(* PLC project fablewhole, LeadShine company LeadSys Studio V3.1.0.0 LeadSysStudio V3.5 SP15 Patch 4 *)
(* stored: creationDateTime 2026-07-10T18:08:29.5976327, modificationDateTime 2026-07-10T18:07:30.2023087 *)

{attribute 'qualified_only'}
{attribute 'strict'}
TYPE E_MachMode : (BOOT := 0, HOMING := 1, READY := 2, RUN := 3, CLEAN := 4, FAULT := 5, ESTOP := 6);
END_TYPE

{attribute 'qualified_only'}
{attribute 'strict'}
TYPE E_Item : (NONE := 0, BEEF := 1, CHICKEN := 2, BACON := 3, PINEAPPLE := 4);
END_TYPE

{attribute 'qualified_only'}
{attribute 'strict'}
TYPE E_GriddleState : (EMPTY := 0, LOADING := 1, COOKING := 2, READY_TO_SCRAPE := 3, SCRAPING := 4, FAULTED := 5);
END_TYPE

{attribute 'qualified_only'}
{attribute 'strict'}
TYPE E_FaultClass : (INFO := 0, QUARANTINE := 1, ZONE_STOP := 2, MACHINE_STOP := 3);
END_TYPE

TYPE ST_Recipe : STRUCT
  item : UINT;  (* E_Item value *)
  cookTimeS : LREAL := 90.0;
  smashDurS : LREAL := 8.0;
  smashPosMm : LREAL := 4.0;  (* platen gap at smash *)
  holdPosMm : LREAL := 6.0;  (* light-contact gap for remainder of cook *)
  platenSetC : LREAL := 200.0;
END_STRUCT;
END_TYPE

TYPE ST_PattyJob : STRUCT
  jobId : UDINT;
  orderId : UDINT;
  item : UINT;
  trayId : UINT;
  griddleId : INT;
  slot : INT;
END_STRUCT;
END_TYPE

TYPE ST_GriddleSts : STRUCT
  state : UINT;  (* E_GriddleState value *)
  item : UINT;
  count : INT;
  cookElapsedS : LREAL;
  batchId : UDINT;
END_STRUCT;
END_TYPE

TYPE ST_TrayInfo : STRUCT
  trayId : UINT;
  item : UINT;
  remaining : INT;
  level : INT;  (* 0..19 *)
  face : INT;  (* 0..1 *)
  inChamber : BOOL;
END_STRUCT;
END_TYPE

TYPE ST_GwCmd : STRUCT
  seq : UINT;
  code : UINT;  (* see GVL_Cfg CMD_* constants *)
  p1 : DINT;
  p2 : DINT;
  p3 : DINT;
  p4 : DINT;
END_STRUCT;
END_TYPE

TYPE ST_GwAck : STRUCT
  seqEcho : UINT;
  busy : BOOL;
  done : BOOL;
  error : BOOL;
  errorId : UDINT;
END_STRUCT;
END_TYPE

TYPE ST_AxisSts : STRUCT
  powered : BOOL;
  homed : BOOL;
  inPos : BOOL;
  actPos : LREAL;
  errorId : UDINT;
END_STRUCT;
END_TYPE

TYPE ST_HeatZone : STRUCT
  setC : LREAL;
  actC : LREAL;
  outPct : LREAL;
  tcOk : BOOL;
  atSet : BOOL;
  enabled : BOOL;
END_STRUCT;
END_TYPE

TYPE ST_Alarm : STRUCT
  id : UDINT;  (* (subsystem<<16) OR code *)
  class : UINT;  (* E_FaultClass value *)
  tsS : UDINT;  (* uptime seconds at raise *)
  active : BOOL;
  acked : BOOL;
END_STRUCT;
END_TYPE

TYPE ST_HaccpRec : STRUCT
  batchId : UDINT;
  item : UINT;
  griddleId : INT;
  platenTopC : LREAL;
  platenBotC : LREAL;
  cookS : LREAL;
  tStartS : UDINT;
  tEndS : UDINT;
  result : UINT;  (* 0=OK 1=QUARANTINE *)
END_STRUCT;
END_TYPE

TYPE ST_MechCmd : STRUCT
  code : UINT;  (* mechanism-local, see GVL_Cfg MCMD_* constants *)
  p1 : LREAL;
  p2 : LREAL;
  p3 : LREAL;
END_STRUCT;
END_TYPE

(* ===== FUNCTION F_Err : UDINT ===== ErrorID encoding: (subsystem << 16) OR code *)
FUNCTION F_Err : UDINT
  VAR_INPUT
    ss : UINT;
    code : UINT;
  END_VAR

                    F_Err := SHL(TO_UDINT(ss), 16) OR TO_UDINT(code);

                  
END_FUNCTION

(* ===== FUNCTION F_RaiseAlarm : BOOL ===== Latch an alarm into GVL_Alm (dedup by id). Returns TRUE if new. *)
FUNCTION F_RaiseAlarm : BOOL
  VAR_INPUT
    id : UDINT;
    class : UINT;  (* E_FaultClass value *)
  END_VAR
  VAR
    i : INT;
  END_VAR

                    F_RaiseAlarm := FALSE;
IF id = 0 THEN RETURN; END_IF
FOR i := 0 TO 63 DO
    IF GVL_Alm.aActive[i].active AND (GVL_Alm.aActive[i].id = id) THEN
        RETURN;                      // already active
    END_IF
END_FOR
FOR i := 0 TO 63 DO
    IF NOT GVL_Alm.aActive[i].active THEN
        GVL_Alm.aActive[i].id     := id;
        GVL_Alm.aActive[i].class  := class;
        GVL_Alm.aActive[i].tsS    := GVL_Sts.uptimeS;
        GVL_Alm.aActive[i].active := TRUE;
        GVL_Alm.aActive[i].acked  := FALSE;
        // history ring
        GVL_Alm.aHistory[GVL_Alm.histHead] := GVL_Alm.aActive[i];
        GVL_Alm.histHead := (GVL_Alm.histHead + 1) MOD 200;
        F_RaiseAlarm := TRUE;
        RETURN;
    END_IF
END_FOR


                  
END_FUNCTION

(* ============================================================ FB_AxisCtrl — single-axis wrapper. The ONLY POU calling MC_*. Runs in T_Motion. One instance per axis, body called EVERY cycle. SIM: internal kinematic model (trapezoid-less: const-vel ramp). REAL: SoftMotion CiA-402 via SM3_Basic. ============================================================ *)
FUNCTION_BLOCK FB_AxisCtrl
  VAR_INPUT
    Sim : BOOL;
    SubsysId : UINT;
    Enable : BOOL;
    HomeExec : BOOL;  (* level; internally edge-latched *)
    MoveExec : BOOL;
    TargetPos : LREAL;
    Vel : LREAL := 100.0;
    Acc : LREAL := 500.0;
    StopExec : BOOL;
    ResetExec : BOOL;
    Abort : BOOL;
    CycleMs : LREAL := 4.0;
    SimHomeS : LREAL := 1.0;  (* sim homing duration *)
  END_VAR
  VAR_IN_OUT
    Axis : AXIS_REF_SM3;
  END_VAR
  VAR_OUTPUT
    Sts : ST_AxisSts;
    Busy : BOOL;
    Done : BOOL;  (* latched until next exec *)
    Error : BOOL;
    ErrorID : UDINT;
  END_VAR
  VAR
    state : INT;  (* 0 idle 1 homing 2 moving 3 stopping *)
    rtHome : R_TRIG;
    rtMove : R_TRIG;
    rtReset : R_TRIG;
    tonTO : TON;
    simPos : LREAL;  (* sim model *)
    simTgt : LREAL;
    simHomeT : LREAL;
    mcPower : MC_Power;  (* real motion FBs *)
    mcHome : MC_Home;
    mcMove : MC_MoveAbsolute;
    mcStop : MC_Stop;
    mcReset : MC_Reset;
    dtS : LREAL;
    stepMax : LREAL;
  END_VAR

                    
dtS := CycleMs / 1000.0;
rtHome(CLK := HomeExec);
rtMove(CLK := MoveExec);
rtReset(CLK := ResetExec);

IF Abort THEN
    state := 0; Busy := FALSE;
    tonTO(IN := FALSE);
END_IF

IF rtReset.Q THEN
    Error := FALSE; ErrorID := 0;
END_IF

IF Sim THEN
    // ---------------- SIMULATION MODEL ----------------
    Sts.powered := Enable;
    CASE state OF
        0: // idle
            IF Enable AND rtHome.Q THEN
                state := 1; simHomeT := 0.0; Busy := TRUE; Done := FALSE;
            ELSIF Enable AND Sts.homed AND rtMove.Q THEN
                simTgt := TargetPos; state := 2; Busy := TRUE; Done := FALSE;
                tonTO(IN := FALSE);
            ELSIF Enable AND (NOT Sts.homed) AND rtMove.Q THEN
                Error := TRUE; ErrorID := F_Err(SubsysId, GVL_Cfg.ERR_NOT_HOMED);
            END_IF
        1: // homing
            simHomeT := simHomeT + dtS;
            IF simHomeT >= SimHomeS THEN
                simPos := 0.0; Sts.homed := TRUE;
                state := 0; Busy := FALSE; Done := TRUE;
            END_IF
        2: // moving: constant-velocity approach
            stepMax := Vel * dtS;
            IF ABS(simTgt - simPos) <= stepMax THEN
                simPos := simTgt;
                state := 0; Busy := FALSE; Done := TRUE;
            ELSIF simTgt > simPos THEN
                simPos := simPos + stepMax;
            ELSE
                simPos := simPos - stepMax;
            END_IF
            tonTO(IN := TRUE, PT := GVL_Cfg.TO_AXIS_MOVE);
            IF tonTO.Q THEN
                state := 0; Busy := FALSE; Error := TRUE;
                ErrorID := F_Err(SubsysId, GVL_Cfg.ERR_TIMEOUT);
            END_IF
    END_CASE
    IF StopExec THEN state := 0; Busy := FALSE; END_IF
    Sts.actPos := simPos;
    Sts.inPos  := (state = 0);
ELSE
    // ---------------- REAL HARDWARE (SoftMotion) ----------------
    mcPower(Axis := Axis, Enable := Enable, bRegulatorOn := Enable, bDriveStart := Enable);
    Sts.powered := mcPower.Status;

    mcHome(Axis := Axis, Execute := (rtHome.Q OR mcHome.Busy) AND NOT Abort, Position := 0.0);
    IF mcHome.Done THEN Sts.homed := TRUE; END_IF

    mcMove(Axis := Axis,
           Execute      := (rtMove.Q OR mcMove.Busy) AND NOT Abort AND NOT StopExec,
           Position     := TargetPos,
           Velocity     := Vel,
           Acceleration := Acc,
           Deceleration := Acc);

    mcStop(Axis := Axis, Execute := StopExec OR Abort, Deceleration := Acc * 2.0);
    mcReset(Axis := Axis, Execute := rtReset.Q);

    Busy := mcHome.Busy OR mcMove.Busy;
    IF mcHome.Done OR mcMove.Done THEN Done := TRUE; END_IF
    IF rtHome.Q OR rtMove.Q THEN Done := FALSE; END_IF

    IF mcMove.Error OR mcHome.Error OR mcPower.Error THEN
        Error := TRUE;
        ErrorID := F_Err(SubsysId, GVL_Cfg.ERR_DRIVE);
        Sts.homed := FALSE;              // demand re-home after drive fault
    END_IF
    Sts.actPos := Axis.fSetPosition;     // TODO: use MC_ReadActualPosition if preferred
    Sts.inPos  := NOT Busy;
END_IF

IF NOT Sts.powered THEN Sts.homed := FALSE; END_IF   // power loss clears homed
Sts.errorId := ErrorID;


                  
END_FUNCTION_BLOCK

(* ============================================================ FB_PidHeater — PI + time-proportioned SSR + TC plausibility. Call every T_App cycle; internal divider executes PI at 100 ms. SIM: first-order plant dT = (gain*out - (T-Tamb)/tau) * dt Independent hardwired thermostat is the REAL protection; the over-temp check here is early warning (INFO/ZONE only). ============================================================ *)
FUNCTION_BLOCK FB_PidHeater
  VAR_INPUT
    Sim : BOOL;
    ZoneId : INT;  (* 0..7 *)
    Enable : BOOL;
    SetC : LREAL := 200.0;
    iTempRaw : INT;  (* 0.1 degC from TC module *)
    StaggerToken : BOOL;  (* may ramp (from FB_HeatBank) *)
    CycleMs : LREAL := 20.0;
  END_VAR
  VAR_OUTPUT
    qSsr : BOOL;
    Zone : ST_HeatZone;
    Error : BOOL;
    ErrorID : UDINT;
  END_VAR
  VAR
    divCnt : INT;
    actC : LREAL;
    lastC : LREAL;
    err : LREAL;
    integ : LREAL;
    outPct : LREAL;
    pwmT : LREAL;
    simC : LREAL := 25.0;
    dtPi : LREAL := 0.1;
    tcFaultCnt : INT;
    SIM_GAIN : LREAL := 3.5;  (* degC/s at 100 % *)
    SIM_TAU : LREAL := 60.0;
    ramping : BOOL;
  END_VAR

                    // ---- acquire temperature ----
IF Sim THEN
    simC := simC + (SIM_GAIN * outPct / 100.0 - (simC - 25.0) / SIM_TAU)
                 * (CycleMs / 1000.0) * GVL_Cfg.SIM_TIME_SCALE;
    actC := simC;
ELSE
    actC := TO_LREAL(iTempRaw) / 10.0;
END_IF

// ---- TC plausibility (real only) ----
IF NOT Sim THEN
    IF (actC < -20.0) OR (actC > 400.0) THEN tcFaultCnt := tcFaultCnt + 1; ELSE tcFaultCnt := 0; END_IF
    IF ABS(actC - lastC) > GVL_Cfg.TC_RATE_MAX * (CycleMs / 1000.0) * 10.0 THEN
        tcFaultCnt := tcFaultCnt + 1;
    END_IF
    IF tcFaultCnt > 25 THEN
        Error := TRUE;
        ErrorID := F_Err(GVL_Cfg.SS_HEAT_0 + TO_UINT(ZoneId), GVL_Cfg.ERR_TC);
    END_IF
END_IF
lastC := actC;

// ---- PI @100 ms ----
divCnt := divCnt + 1;
IF divCnt >= 5 THEN
    divCnt := 0;
    ramping := (SetC - actC) > 20.0;
    IF Enable AND NOT Error AND (StaggerToken OR NOT ramping) THEN
        err := SetC - actC;
        integ := LIMIT(0.0, integ + err * GVL_Cfg.HEAT_KI * dtPi * 100.0, 100.0);
        outPct := LIMIT(0.0, GVL_Cfg.HEAT_KP * err + integ, 100.0);
    ELSE
        outPct := 0.0; integ := 0.0;
    END_IF
END_IF

// ---- time-proportioned SSR ----
pwmT := pwmT + CycleMs;
IF pwmT >= GVL_Cfg.PWM_WINDOW_MS THEN pwmT := 0.0; END_IF
qSsr := Enable AND NOT Error AND (pwmT < outPct / 100.0 * GVL_Cfg.PWM_WINDOW_MS);

Zone.setC := SetC;   Zone.actC := actC;   Zone.outPct := outPct;
Zone.tcOk := NOT Error;
Zone.atSet := ABS(SetC - actC) <= GVL_Cfg.HEAT_AT_BAND;
Zone.enabled := Enable;


                  
END_FUNCTION_BLOCK

(* ============================================================ FB_PneuActuator — valve + 2 reed/prox sensors + timeout. Cmd TRUE = extend/open, FALSE = retract/close. Runs in T_App. SIM: sensors flip after SIM_TRAVEL_S. ============================================================ *)
FUNCTION_BLOCK FB_PneuActuator
  VAR_INPUT
    Sim : BOOL;
    SubsysId : UINT;
    Cmd : BOOL;
    iExtended : BOOL;
    iRetracted : BOOL;
    CycleMs : LREAL := 20.0;
  END_VAR
  VAR_OUTPUT
    qValve : BOOL;
    Extended : BOOL;
    Retracted : BOOL;
    Moving : BOOL;
    Error : BOOL;
    ErrorID : UDINT;
  END_VAR
  VAR
    tonTO : TON;
    lastCmd : BOOL;
    simT : LREAL;
    simExt : BOOL;
    SIM_TRAVEL_S : LREAL := 0.3;
    extEff : BOOL;
    retEff : BOOL;
  END_VAR

                    
qValve := Cmd;
IF Cmd <> lastCmd THEN
    simT := 0.0;
    lastCmd := Cmd;
END_IF

IF Sim THEN
    simT := simT + CycleMs / 1000.0;
    IF simT >= SIM_TRAVEL_S THEN simExt := Cmd; END_IF
    extEff := simExt;  retEff := NOT simExt;
ELSE
    extEff := iExtended; retEff := iRetracted;
END_IF

IF extEff AND retEff THEN                 // both sensors -> wiring fault
    Error := TRUE; ErrorID := F_Err(SubsysId, GVL_Cfg.ERR_SENSOR);
END_IF

Extended  := extEff AND NOT retEff;
Retracted := retEff AND NOT extEff;
Moving    := NOT Extended AND NOT Retracted;

tonTO(IN := (Cmd AND NOT Extended) OR (NOT Cmd AND NOT Retracted), PT := GVL_Cfg.TO_PNEU);
IF tonTO.Q THEN
    Error := TRUE; ErrorID := F_Err(SubsysId, GVL_Cfg.ERR_TIMEOUT);
END_IF


                  
END_FUNCTION_BLOCK

(* ============================================================ FB_PressDrive — CS2RS in PR mode, DI-trigger control. Validated pattern from the gantry test project: - set path-select DOs, wait one cycle, raise CTRG and HOLD it until InPos confirms (never a single-scan pulse) - InPos handshake = "saw moving" (InPos drops, then returns) Modbus RTU monitoring (position/alarm) is DIAGNOSTIC ONLY and added at migration (stub hooks below). Runs in T_App (20 ms). PR paths (configure in drive, MIGRATION_GUIDE step 4): path 0 = OPEN position, path 1 = SMASH pos, path 2 = HOLD pos ============================================================ *)
FUNCTION_BLOCK FB_PressDrive
  VAR_INPUT
    Sim : BOOL;
    SubsysId : UINT;
    Enable : BOOL;
    PathExec : BOOL;  (* edge latches PathNo *)
    PathNo : INT;  (* 0..2 *)
    Abort : BOOL;
    iInPos : BOOL;  (* from drive DO (via IoMap) *)
    iAlarm : BOOL;
    CycleMs : LREAL := 20.0;
    OpenPosMm : LREAL := 60.0;  (* path 0 *)
    SmashPosMm : LREAL := 4.0;  (* path 1 *)
    HoldPosMm : LREAL := 6.0;  (* path 2 *)
    WriteParams : BOOL;  (* edge: push the 3 positions to the drive *)
    MbWrDone : BOOL;  (* transport confirms last write *)
    MbWrErr : BOOL;  (* transport reports failure *)
  END_VAR
  VAR_OUTPUT
    qSel0 : BOOL;
    qSel1 : BOOL;
    qCtrg : BOOL;
    qEnable : BOOL;
    Busy : BOOL;
    Done : BOOL;
    Error : BOOL;
    ErrorID : UDINT;
    ActPath : INT := -1;
    ParamsValid : BOOL;  (* drive path table matches last written values *)
    ParamBusy : BOOL;
    ParamErr : BOOL;
    MbPath : INT;  (* which PR path's position is being written (0..2) *)
    MbValH : WORD;  (* position high word *)
    MbValL : WORD;  (* position low word *)
    MbWrExec : BOOL;  (* held TRUE until MbWrDone/MbWrErr *)
  END_VAR
  VAR
    state : INT;
    rtExec : R_TRIG;
    latched : INT;
    sawMoving : BOOL;
    tonTO : TON;
    inPosEff : BOOL;
    simTimer : LREAL;  (* sim *)
    SIM_TRAVEL_S : LREAL := 0.8;
    rtWr : R_TRIG;  (* param write channel *)
    pStep : INT;
    pRetry : INT;
    P_MAX_RETRY : INT := 3;
    shadowOpen : LREAL;  (* last values confirmed in drive *)
    shadowSmash : LREAL;  (* last values confirmed in drive *)
    shadowHold : LREAL;  (* last values confirmed in drive *)
    pInit : BOOL;  (* at least one successful full push done *)
    pIdx : INT;  (* 0..2: one write per PR path (posH+posL together) *)
    pPosMm : LREAL;
    pPulses : DINT;
    tonMb : TON;  (* per-transaction timeout *)
  END_VAR

                    rtExec(CLK := PathExec);
qEnable := Enable;

// effective InPos: sim model or hardware input
IF Sim THEN
    inPosEff := (state <> 3) OR (simTimer >= SIM_TRAVEL_S);
ELSE
    inPosEff := iInPos;
END_IF

IF Abort THEN
    state := 0; Busy := FALSE; qCtrg := FALSE;
    tonTO(IN := FALSE);
END_IF

IF (NOT Sim) AND iAlarm THEN
    Error := TRUE; ErrorID := F_Err(SubsysId, GVL_Cfg.ERR_DRIVE);
    state := 0; Busy := FALSE; qCtrg := FALSE;
    pInit := FALSE;   // drive may have power-cycled: RAM PR table reverts to
                      // EEPROM, so force a full re-push on the next profile
END_IF

CASE state OF
    0: // idle
        qCtrg := FALSE;
        IF Enable AND rtExec.Q AND (PathNo >= 0) AND (PathNo <= 2) THEN
            latched := PathNo;
            qSel0 := (latched MOD 2) = 1;
            qSel1 := ((latched / 2) MOD 2) = 1;
            state := 1; Busy := TRUE; Done := FALSE;
            sawMoving := FALSE; simTimer := 0.0;
            tonTO(IN := FALSE);
        END_IF
    1: // one full cycle DO settle before CTRG (drive DI filter)
        state := 3;
        qCtrg := TRUE;                     // held high for whole move
    3: // executing: wait saw-moving handshake
        simTimer := simTimer + CycleMs / 1000.0;
        IF NOT inPosEff THEN sawMoving := TRUE; END_IF
        tonTO(IN := TRUE, PT := GVL_Cfg.TO_PRESS);
        IF inPosEff AND (sawMoving OR (Sim AND simTimer >= SIM_TRAVEL_S)) THEN
            qCtrg := FALSE; ActPath := latched;
            state := 0; Busy := FALSE; Done := TRUE;
            tonTO(IN := FALSE);
        ELSIF tonTO.Q THEN
            qCtrg := FALSE;
            state := 0; Busy := FALSE; Error := TRUE;
            ErrorID := F_Err(SubsysId, GVL_Cfg.ERR_TIMEOUT);
        END_IF
END_CASE

// ============================================================
// PR path table parameter writer (positions only; motion stays DI).
// SIM: accepted instantly. HARDWARE: closed-loop Modbus RTU write ->
// readback verify -> retry (pattern proven on the old Z-axis rig).
// Only call while press idle; FB_Press guarantees this.
// ============================================================
rtWr(CLK := WriteParams);
IF rtWr.Q AND (pStep = 0) THEN
    ParamsValid := FALSE; ParamErr := FALSE; ParamBusy := TRUE;
    pRetry := 0; pStep := 1;
END_IF

CASE pStep OF
    0: ;
    1: // route: skip if drive already holds these values
        IF pInit AND (OpenPosMm = shadowOpen) AND (SmashPosMm = shadowSmash)
                 AND (HoldPosMm = shadowHold) THEN
            ParamsValid := TRUE; ParamBusy := FALSE; pStep := 0;
        ELSIF Sim THEN
            // simulation: accept instantly
            shadowOpen := OpenPosMm; shadowSmash := SmashPosMm; shadowHold := HoldPosMm;
            pInit := TRUE;
            ParamsValid := TRUE; ParamBusy := FALSE; pStep := 0;
        ELSE
            pIdx := 0; pStep := 2;                        // real Modbus push, path by path
        END_IF
    2: // compose path write pIdx (posH+posL in one write-multiple transaction)
        CASE pIdx OF
            0: pPosMm := OpenPosMm;
            1: pPosMm := SmashPosMm;
            2: pPosMm := HoldPosMm;
        END_CASE
        pPulses := TO_DINT(pPosMm * GVL_Cfg.PRESS_PULSES_PER_MM);
        MbPath := pIdx;
        MbValH := TO_WORD(SHR(TO_DWORD(pPulses), 16) AND 16#FFFF);
        MbValL := TO_WORD(TO_DWORD(pPulses) AND 16#FFFF);
        MbWrExec := TRUE; tonMb(IN := FALSE);
        pStep := 3;
    3: // wait channel ack (glue reflects the NetworkConfig channel done/error)
        tonMb(IN := TRUE, PT := T#1S);
        IF MbWrDone THEN
            MbWrExec := FALSE; tonMb(IN := FALSE); pRetry := 0;
            pIdx := pIdx + 1;
            IF pIdx > 2 THEN
                shadowOpen := OpenPosMm; shadowSmash := SmashPosMm; shadowHold := HoldPosMm;
                pInit := TRUE;
                ParamsValid := TRUE; ParamBusy := FALSE; pStep := 0;
            ELSE
                pStep := 2;                               // next path (fresh trigger edge)
            END_IF
        ELSIF MbWrErr OR tonMb.Q THEN
            MbWrExec := FALSE; tonMb(IN := FALSE);
            pRetry := pRetry + 1;
            IF pRetry > P_MAX_RETRY THEN
                ParamErr := TRUE; ParamBusy := FALSE; pStep := 0;
            ELSE
                pStep := 2;                               // resend same path
            END_IF
        END_IF
END_CASE

// TODO(MIGRATION): background Modbus RTU poll <=2 Hz for ActPosMm +
// AlarmCode; failure raises INFO alarm only, never blocks motion.

                  
END_FUNCTION_BLOCK

(* ============================================================ FB_SensorIn — debounced digital input. SIM: output follows SimValue directly. ============================================================ *)
FUNCTION_BLOCK FB_SensorIn
  VAR_INPUT
    Sim : BOOL;
    SimValue : BOOL;
    iRaw : BOOL;
    DebounceMs : LREAL := 40.0;
    CycleMs : LREAL := 20.0;
  END_VAR
  VAR_OUTPUT
    Q : BOOL;
  END_VAR
  VAR
    acc : LREAL;
    lastRaw : BOOL;
  END_VAR

                    IF Sim THEN
    Q := SimValue;
ELSE
    IF iRaw = lastRaw THEN
        acc := acc + CycleMs;
        IF acc >= DebounceMs THEN Q := iRaw; END_IF
    ELSE
        acc := 0.0;
        lastRaw := iRaw;
    END_IF
END_IF


                  
END_FUNCTION_BLOCK

(* ============================================================ FB_VfdIndex — carousel indexing: VFD run/dir + encoder + pin. Pin actuator is external (FB_PneuActuator); this FB commands it via PinCmd and reads PinExtended/PinRetracted. Sequence: retract pin -> rotate (fast->creep) -> stop in window -> extend pin -> verify pin + encoder plausibility. Runs in T_App. SIM: integrates encoder; home prox modeled. ============================================================ *)
FUNCTION_BLOCK FB_VfdIndex
  VAR_INPUT
    Sim : BOOL;
    SubsysId : UINT;
    Enable : BOOL;
    HomeExec : BOOL;
    GotoExec : BOOL;
    TargetStation : INT;
    Bidirectional : BOOL;
    Abort : BOOL;
    iEnc : DINT;
    iHomeProx : BOOL;
    PinExtended : BOOL;
    PinRetracted : BOOL;
    CycleMs : LREAL := 20.0;
  END_VAR
  VAR_OUTPUT
    qFwd : BOOL;
    qRev : BOOL;
    qSpeed : INT;
    PinCmd : BOOL := TRUE;  (* TRUE = extend (locked at rest) *)
    ActStation : INT := -1;
    Homed : BOOL;
    Busy : BOOL;
    Done : BOOL;
    Error : BOOL;
    ErrorID : UDINT;
  END_VAR
  VAR
    state : INT;
    rtHome : R_TRIG;
    rtGoto : R_TRIG;
    tonTO : TON;
    encEff : DINT;
    homeEff : BOOL;
    encZero : DINT;  (* count value at station 0 *)
    tgtCounts : DINT;
    diff : DINT;
    cps : DINT;  (* counts per station *)
    fwdDir : BOOL;
    goingHome : BOOL;
    simEnc : DINT;
    stepC : DINT;
  END_VAR

                    cps := GVL_Cfg.ENC_CPR / TO_DINT(GVL_Cfg.STATIONS);
rtHome(CLK := HomeExec);
rtGoto(CLK := GotoExec);

// ------- feedback source -------
IF Sim THEN
    IF qFwd THEN
        stepC := TO_DINT(TO_LREAL(qSpeed) * CycleMs / 20.0);
        simEnc := simEnc + MAX(stepC, 1);
    ELSIF qRev THEN
        stepC := TO_DINT(TO_LREAL(qSpeed) * CycleMs / 20.0);
        simEnc := simEnc - MAX(stepC, 1);
    END_IF
    encEff  := simEnc;
    homeEff := ((simEnc MOD GVL_Cfg.ENC_CPR) + GVL_Cfg.ENC_CPR) MOD GVL_Cfg.ENC_CPR < 60;
ELSE
    encEff  := iEnc;
    homeEff := iHomeProx;
END_IF

IF Abort THEN
    qFwd := FALSE; qRev := FALSE; qSpeed := 0;
    state := 0; Busy := FALSE; tonTO(IN := FALSE);
END_IF

CASE state OF
    0: // idle (pin extended = locked)
        qFwd := FALSE; qRev := FALSE; qSpeed := 0;
        IF Enable AND rtHome.Q THEN
            goingHome := TRUE; state := 10; Busy := TRUE; Done := FALSE;
        ELSIF Enable AND Homed AND rtGoto.Q THEN
            IF (TargetStation < 0) OR (TargetStation >= GVL_Cfg.STATIONS) THEN
                Error := TRUE; ErrorID := F_Err(SubsysId, GVL_Cfg.ERR_BAD_CMD);
            ELSIF TargetStation = ActStation THEN
                Done := TRUE;
            ELSE
                goingHome := FALSE; state := 10; Busy := TRUE; Done := FALSE;
            END_IF
        END_IF

    10: // retract pin
        PinCmd := FALSE;
        tonTO(IN := TRUE, PT := GVL_Cfg.TO_PNEU);
        IF PinRetracted THEN
            tonTO(IN := FALSE); state := 20;
        ELSIF tonTO.Q THEN
            state := 90; ErrorID := F_Err(SubsysId, GVL_Cfg.ERR_PIN);
        END_IF

    20: // rotate
        IF goingHome THEN
            qFwd := TRUE; qSpeed := GVL_Cfg.IDX_SPEED_CREEP;
            tonTO(IN := TRUE, PT := GVL_Cfg.TO_INDEX);
            IF homeEff THEN
                qFwd := FALSE; qSpeed := 0;
                encZero := encEff;
                tonTO(IN := FALSE); state := 30;
            ELSIF tonTO.Q THEN
                state := 90; ErrorID := F_Err(SubsysId, GVL_Cfg.ERR_TIMEOUT);
            END_IF
        ELSE
            tgtCounts := encZero + TO_DINT(TargetStation) * cps;
            diff := tgtCounts - encEff;
            IF Bidirectional THEN
                // shortest signed path within one revolution
                diff := ((diff MOD GVL_Cfg.ENC_CPR) + GVL_Cfg.ENC_CPR) MOD GVL_Cfg.ENC_CPR;
                IF diff > GVL_Cfg.ENC_CPR / 2 THEN diff := diff - GVL_Cfg.ENC_CPR; END_IF
            ELSE
                diff := ((diff MOD GVL_Cfg.ENC_CPR) + GVL_Cfg.ENC_CPR) MOD GVL_Cfg.ENC_CPR;
            END_IF
            fwdDir := diff >= 0;
            qFwd := fwdDir AND (ABS(diff) > GVL_Cfg.IDX_STOP_WIN);
            qRev := (NOT fwdDir) AND (ABS(diff) > GVL_Cfg.IDX_STOP_WIN);
            IF ABS(diff) > GVL_Cfg.IDX_DECEL_WIN THEN
                qSpeed := GVL_Cfg.IDX_SPEED_FAST;
            ELSE
                qSpeed := GVL_Cfg.IDX_SPEED_CREEP;
            END_IF
            tonTO(IN := TRUE, PT := GVL_Cfg.TO_INDEX);
            IF ABS(diff) <= GVL_Cfg.IDX_STOP_WIN THEN
                qFwd := FALSE; qRev := FALSE; qSpeed := 0;
                tonTO(IN := FALSE); state := 30;
            ELSIF tonTO.Q THEN
                state := 90; ErrorID := F_Err(SubsysId, GVL_Cfg.ERR_TIMEOUT);
            END_IF
        END_IF

    30: // extend pin + verify
        PinCmd := TRUE;
        tonTO(IN := TRUE, PT := GVL_Cfg.TO_PNEU);
        IF PinExtended THEN
            tonTO(IN := FALSE);
            IF goingHome THEN
                Homed := TRUE; ActStation := 0;
            ELSE
                // encoder-vs-pin plausibility
                diff := (((encEff - encZero) MOD GVL_Cfg.ENC_CPR) + GVL_Cfg.ENC_CPR) MOD GVL_Cfg.ENC_CPR;
                IF ABS(diff - TO_DINT(TargetStation) * cps) > GVL_Cfg.IDX_VERIFY_WIN THEN
                    state := 90; ErrorID := F_Err(SubsysId, GVL_Cfg.ERR_PIN);
                    Homed := FALSE;                    // demand re-home
                    RETURN;
                END_IF
                ActStation := TargetStation;
            END_IF
            state := 0; Busy := FALSE; Done := TRUE;
        ELSIF tonTO.Q THEN
            state := 90; ErrorID := F_Err(SubsysId, GVL_Cfg.ERR_PIN);
        END_IF

    90: // fault
        qFwd := FALSE; qRev := FALSE; qSpeed := 0;
        Busy := FALSE; Error := TRUE;
        state := 0;
END_CASE


                  
END_FUNCTION_BLOCK

(* ============================================================ FB_Airlock — chamber gate mutual exclusion. Requests are LEVELS; the FB grants at most one open door, closing the other first. ChamberSealed = both confirmed closed. Runs in T_App. DoorFridge = fridge-side gate, DoorChamber = griddle-side gate. ============================================================ *)
FUNCTION_BLOCK FB_Airlock
  VAR_INPUT
    Enable : BOOL;
    ReqFridgeOpen : BOOL;
    ReqChamberOpen : BOOL;
    Abort : BOOL;
  END_VAR
  VAR_IN_OUT
    DoorFridge : FB_PneuActuator;
    DoorChamber : FB_PneuActuator;
  END_VAR
  VAR_OUTPUT
    FridgeOpen : BOOL;
    ChamberOpen : BOOL;
    ChamberSealed : BOOL;
    Busy : BOOL;
    Error : BOOL;
    ErrorID : UDINT;
  END_VAR
  VAR
    wantF : BOOL;
    wantC : BOOL;
  END_VAR

                    wantF := Enable AND ReqFridgeOpen AND NOT Abort;
wantC := Enable AND ReqChamberOpen AND NOT Abort;

// mutual exclusion: fridge side has priority; never open one until
// the other is CONFIRMED retracted (closed)
IF wantF AND wantC THEN wantC := FALSE; END_IF
DoorFridge.Cmd  := wantF AND DoorChamber.Retracted;
DoorChamber.Cmd := wantC AND DoorFridge.Retracted;

FridgeOpen    := DoorFridge.Extended;
ChamberOpen   := DoorChamber.Extended;
ChamberSealed := DoorFridge.Retracted AND DoorChamber.Retracted;
Busy := (wantF AND NOT FridgeOpen) OR (wantC AND NOT ChamberOpen)
     OR ((NOT wantF) AND NOT DoorFridge.Retracted)
     OR ((NOT wantC) AND NOT DoorChamber.Retracted);

IF DoorFridge.Error OR DoorChamber.Error THEN
    Error := TRUE;
    ErrorID := F_Err(GVL_Cfg.SS_AIRLOCK, GVL_Cfg.ERR_TIMEOUT);
ELSE
    Error := FALSE; ErrorID := 0;
END_IF

// hard invariant — must never trip, in sim or real
IF FridgeOpen AND ChamberOpen THEN
    Error := TRUE;
    ErrorID := F_Err(GVL_Cfg.SS_AIRLOCK, GVL_Cfg.ERR_INTERLOCK);
END_IF


                  
END_FUNCTION_BLOCK

(* ============================================================ FB_Fork — tray fetch/return, 2 axes + fail-safe brake. Commands: MCMD_HOME, MCMD_FETCH(p1=level), MCMD_RETURN(p1=level). Fetch: Z to level -> tele out -> micro-lift (release stacking lock) -> tele in (tray drawn into chamber). Return: Z to level+micro -> tele out -> micro-drop (re-engage lock) -> tele in. Brake: qBrakeRelease TRUE only while Z powered & healthy; a feedback mismatch is MACHINE_STOP class. Runs in T_Motion. ============================================================ *)
FUNCTION_BLOCK FB_Fork
  VAR_INPUT
    Enable : BOOL;
    Cmd : ST_MechCmd;
    CmdExec : BOOL;
    Abort : BOOL;
    Sim : BOOL;
    iBrakeOk : BOOL;
    iTrayPresent : BOOL;
  END_VAR
  VAR_IN_OUT
    AxZ : FB_AxisCtrl;
    AxT : FB_AxisCtrl;  (* telescope *)
  END_VAR
  VAR_OUTPUT
    qBrakeRelease : BOOL;
    TrayHeld : BOOL;
    Busy : BOOL;
    Done : BOOL;
    Error : BOOL;
    ErrorID : UDINT;
    State : UINT;
    Homed : BOOL;
  END_VAR
  VAR
    iSt : INT;
    rtExec : R_TRIG;
    level : INT;
    zBase : LREAL;
    fetching : BOOL;
    brakeChk : TON;
    tonTO : TON;
    trayEff : BOOL;
  END_VAR

                    rtExec(CLK := CmdExec);
trayEff := (Sim AND TrayHeld) OR ((NOT Sim) AND iTrayPresent);

// brake proving: release demand vs feedback
qBrakeRelease := Enable AND AxZ.Sts.powered AND NOT Abort AND NOT Error;
brakeChk(IN := (NOT Sim) AND (qBrakeRelease <> iBrakeOk), PT := T#500MS);
IF brakeChk.Q THEN
    Error := TRUE;
    ErrorID := F_Err(GVL_Cfg.SS_FORK_Z, GVL_Cfg.ERR_DRIVE);   // MACHINE_STOP via PRG_Alarms map
END_IF

IF Abort THEN
    iSt := 0; Busy := FALSE;
    AxZ.MoveExec := FALSE; AxT.MoveExec := FALSE;
    AxZ.HomeExec := FALSE; AxT.HomeExec := FALSE;
END_IF
Homed := AxZ.Sts.homed AND AxT.Sts.homed;

tonTO(IN := Busy, PT := GVL_Cfg.TO_MECH);
IF tonTO.Q AND Busy THEN
    iSt := 0; Busy := FALSE; Error := TRUE;
    ErrorID := F_Err(GVL_Cfg.SS_FORK, GVL_Cfg.ERR_TIMEOUT);
END_IF

CASE iSt OF
    0:
        IF Enable AND rtExec.Q AND NOT Error THEN
            Done := FALSE; ErrorID := 0;
            CASE Cmd.code OF
                1:  (* MCMD_HOME *)  iSt := 10; Busy := TRUE;
                20, 21: (* MCMD_FETCH / MCMD_RETURN *)
                    level := TO_INT(Cmd.p1);
                    IF (level < 0) OR (level >= GVL_Cfg.TRAY_LEVELS) THEN
                        Error := TRUE; ErrorID := F_Err(GVL_Cfg.SS_FORK, GVL_Cfg.ERR_BAD_CMD);
                    ELSE
                        fetching := (Cmd.code = GVL_Cfg.MCMD_FETCH);  // constant compare OK outside CASE labels
                        zBase := GVL_Cfg.FORK_Z0 + TO_LREAL(level) * GVL_Cfg.FORK_LEVEL_H;
                        iSt := 20; Busy := TRUE;
                    END_IF
            ELSE
                Error := TRUE; ErrorID := F_Err(GVL_Cfg.SS_FORK, GVL_Cfg.ERR_BAD_CMD);
            END_CASE
        END_IF
    10: // HOME: telescope retract first, then Z
        AxT.HomeExec := TRUE;
        IF AxT.Sts.homed THEN AxT.HomeExec := FALSE; iSt := 11; END_IF
    11:
        AxZ.HomeExec := TRUE;
        IF AxZ.Sts.homed THEN
            AxZ.HomeExec := FALSE; iSt := 0; Busy := FALSE; Done := TRUE;
        END_IF
    20: // Z to level (fetch: exact; return: +microlift so tray clears)
        IF fetching THEN AxZ.TargetPos := zBase;
        ELSE AxZ.TargetPos := zBase + GVL_Cfg.FORK_MICROLIFT; END_IF
        AxZ.Vel := GVL_Cfg.F_VEL; AxZ.Acc := GVL_Cfg.F_ACC;
        AxZ.MoveExec := TRUE;
        IF AxZ.Done THEN AxZ.MoveExec := FALSE; iSt := 21; END_IF
        IF AxZ.Error THEN iSt := 90; END_IF
    21: // telescope out
        AxT.TargetPos := GVL_Cfg.FORK_TELE_OUT; AxT.Vel := GVL_Cfg.F_VEL; AxT.Acc := GVL_Cfg.F_ACC;
        AxT.MoveExec := TRUE;
        IF AxT.Done THEN AxT.MoveExec := FALSE; iSt := 22; END_IF
        IF AxT.Error THEN iSt := 90; END_IF
    22: // micro-lift (fetch) or micro-drop (return)
        IF fetching THEN AxZ.TargetPos := zBase + GVL_Cfg.FORK_MICROLIFT;
        ELSE AxZ.TargetPos := zBase; END_IF
        AxZ.MoveExec := TRUE;
        IF AxZ.Done THEN AxZ.MoveExec := FALSE; iSt := 23; END_IF
        IF AxZ.Error THEN iSt := 90; END_IF
    23: // telescope in
        AxT.TargetPos := GVL_Cfg.FORK_TELE_IN; AxT.MoveExec := TRUE;
        IF AxT.Done THEN
            AxT.MoveExec := FALSE;
            IF fetching THEN
                TrayHeld := TRUE;
                IF Sim OR trayEff THEN
                    iSt := 0; Busy := FALSE; Done := TRUE;
                ELSE
                    TrayHeld := FALSE;
                    iSt := 0; Busy := FALSE; Error := TRUE;
                    ErrorID := F_Err(GVL_Cfg.SS_FORK, GVL_Cfg.ERR_SENSOR);  // tray not present
                END_IF
            ELSE
                TrayHeld := FALSE;
                iSt := 0; Busy := FALSE; Done := TRUE;
            END_IF
        END_IF
        IF AxT.Error THEN iSt := 90; END_IF
    90:
        AxZ.MoveExec := FALSE; AxT.MoveExec := FALSE;
        IF ErrorID = 0 THEN
            IF AxZ.Error THEN ErrorID := AxZ.ErrorID;
            ELSIF AxT.Error THEN ErrorID := AxT.ErrorID;
            ELSE ErrorID := F_Err(GVL_Cfg.SS_FORK, GVL_Cfg.ERR_DRIVE); END_IF
        END_IF
        iSt := 0; Busy := FALSE; Error := TRUE;
END_CASE
State := TO_UINT(iSt);

                  
END_FUNCTION_BLOCK

(* ============================================================ FB_FridgeCarousel — tray column indexing (2 faces). Identical pattern to the griddle carousel, no rotation permissive beyond fork-retracted (wired by caller as Permissive). Unidirectional is acceptable here. Runs in T_App. ============================================================ *)
FUNCTION_BLOCK FB_FridgeCarousel
  VAR_INPUT
    Enable : BOOL;
    HomeExec : BOOL;
    GotoExec : BOOL;
    TargetFace : INT;  (* 0..1 mapped to stations 0 / STATIONS/2 *)
    Permissive : BOOL;  (* fork telescope retracted *)
    Abort : BOOL;
  END_VAR
  VAR_IN_OUT
    Vfd : FB_VfdIndex;
    Pin : FB_PneuActuator;
  END_VAR
  VAR_OUTPUT
    ActFace : INT;
    Homed : BOOL;
    Busy : BOOL;
    Done : BOOL;
    Error : BOOL;
    ErrorID : UDINT;
  END_VAR
  VAR
    rtGoto : R_TRIG;
  END_VAR

                    rtGoto(CLK := GotoExec);
IF rtGoto.Q AND NOT Permissive THEN
    Error := TRUE;
    ErrorID := F_Err(GVL_Cfg.SS_FRIDGE_CAR, GVL_Cfg.ERR_INTERLOCK);
END_IF

Pin.Cmd          := Vfd.PinCmd;
Vfd.PinExtended  := Pin.Extended;
Vfd.PinRetracted := Pin.Retracted;

Vfd.Enable   := Enable;
Vfd.Abort    := Abort;
Vfd.HomeExec := HomeExec;
Vfd.GotoExec := GotoExec AND Permissive;
Vfd.TargetStation := TargetFace * (GVL_Cfg.STATIONS / 2);
Vfd.Bidirectional := FALSE;

IF Vfd.ActStation = 0 THEN ActFace := 0;
ELSIF Vfd.ActStation = GVL_Cfg.STATIONS / 2 THEN ActFace := 1;
ELSE ActFace := -1; END_IF
Homed := Vfd.Homed;
Busy  := Vfd.Busy;
Done  := Vfd.Done;
IF Vfd.Error OR Pin.Error THEN
    Error := TRUE;
    IF Vfd.Error THEN ErrorID := Vfd.ErrorID; ELSE ErrorID := Pin.ErrorID; END_IF
END_IF


                  
END_FUNCTION_BLOCK

(* ============================================================ FB_Gantry — pick/place mechanism. Standard interface (spec sec.12). Owns sequencing only; axis FB bodies are called in PRG_Motion. Commands: MCMD_HOME, MCMD_PICK(p1=trayIdx 0..23), MCMD_PLACE(p1=slot 0..5), MCMD_PARK, MCMD_SANITIZE. Coordinated XY = simultaneous X + theta targets (v1; swap to interpolated transform after IK validation without touching callers — see method note in spec 9.1). Runs in T_Motion. ============================================================ *)
FUNCTION_BLOCK FB_Gantry
  VAR_INPUT
    Enable : BOOL;
    Cmd : ST_MechCmd;
    CmdExec : BOOL;
    Abort : BOOL;
    Sim : BOOL;
  END_VAR
  VAR_IN_OUT
    AxX : FB_AxisCtrl;
    AxT : FB_AxisCtrl;
    AxZ : FB_AxisCtrl;
    Grip : FB_Gripper;
    IK : FB_IKTransform;
  END_VAR
  VAR_OUTPUT
    Busy : BOOL;
    Done : BOOL;
    Error : BOOL;
    ErrorID : UDINT;
    State : UINT;
    Homed : BOOL;
    Parked : BOOL;
  END_VAR
  VAR
    iSt : INT;
    rtExec : R_TRIG;
    cmdL : ST_MechCmd;
    tgtX : LREAL;
    tgtY : LREAL;
    zTarget : LREAL;
    idx : INT;
    row : INT;
    col : INT;
    tonTO : TON;
  END_VAR

                    
rtExec(CLK := CmdExec);

IF Abort THEN
    iSt := 0; Busy := FALSE;
    AxX.MoveExec := FALSE; AxT.MoveExec := FALSE; AxZ.MoveExec := FALSE;
    AxX.HomeExec := FALSE; AxT.HomeExec := FALSE; AxZ.HomeExec := FALSE;
    tonTO(IN := FALSE);
END_IF

Homed  := AxX.Sts.homed AND AxT.Sts.homed AND AxZ.Sts.homed;
Parked := Homed AND (iSt = 0) AND (ABS(AxX.Sts.actPos - GVL_Cfg.GX_PARK) < 2.0);

tonTO(IN := Busy, PT := GVL_Cfg.TO_MECH);
IF tonTO.Q AND Busy THEN
    iSt := 0; Busy := FALSE; Error := TRUE;
    ErrorID := F_Err(GVL_Cfg.SS_GANTRY, GVL_Cfg.ERR_TIMEOUT);
END_IF

CASE iSt OF
    0: // IDLE — accept command
        IF Enable AND rtExec.Q THEN
            cmdL := Cmd; Done := FALSE; Error := FALSE; ErrorID := 0;
            CASE cmdL.code OF
                1:  (* MCMD_HOME *)     iSt := 10; Busy := TRUE;
                10: (* MCMD_PICK *)
                    idx := TO_INT(cmdL.p1);
                    row := idx / GVL_Cfg.TRAY_COLS;  col := idx MOD GVL_Cfg.TRAY_COLS;
                    tgtX := GVL_Cfg.PICK_BASE_X + TO_LREAL(col) * GVL_Cfg.PICK_SPACING_X + GVL_Par.pickOffsetX;
                    tgtY := GVL_Cfg.PICK_BASE_Y + TO_LREAL(row) * GVL_Cfg.PICK_SPACING_Y + GVL_Par.pickOffsetY;
                    zTarget := GVL_Cfg.GZ_PICK;
                    iSt := 20; Busy := TRUE;
                11: (* MCMD_PLACE *)
                    idx := TO_INT(cmdL.p1);
                    row := idx / GVL_Cfg.PLACE_COLS; col := idx MOD GVL_Cfg.PLACE_COLS;
                    tgtX := GVL_Cfg.PLACE_BASE_X + TO_LREAL(col) * GVL_Cfg.PLACE_SPC_X + GVL_Par.placeOffsetX;
                    tgtY := GVL_Cfg.PLACE_BASE_Y + TO_LREAL(row) * GVL_Cfg.PLACE_SPC_Y + GVL_Par.placeOffsetY;
                    zTarget := GVL_Cfg.GZ_PLACE;
                    iSt := 20; Busy := TRUE;
                2:  (* MCMD_PARK *)
                    tgtX := GVL_Cfg.GX_PARK; tgtY := GVL_Cfg.ARM_LEN * 0.0;
                    iSt := 60; Busy := TRUE;
                13: (* MCMD_SANITIZE *)
                    tgtX := GVL_Cfg.GX_MAX;  tgtY := 0.0;    // wash-station pose TODO
                    iSt := 60; Busy := TRUE;
            ELSE
                Error := TRUE; ErrorID := F_Err(GVL_Cfg.SS_GANTRY, GVL_Cfg.ERR_BAD_CMD);
            END_CASE
        END_IF

    10: // HOME: Z up first, then theta safe, then X (collision-safe)
        AxZ.HomeExec := TRUE;
        IF AxZ.Sts.homed THEN AxZ.HomeExec := FALSE; iSt := 11; END_IF
    11:
        AxT.HomeExec := TRUE;
        IF AxT.Sts.homed THEN AxT.HomeExec := FALSE; iSt := 12; END_IF
    12:
        AxX.HomeExec := TRUE;
        IF AxX.Sts.homed THEN
            AxX.HomeExec := FALSE;
            iSt := 0; Busy := FALSE; Done := TRUE;
        END_IF

    20: // PICK/PLACE step 1: Z up
        AxZ.TargetPos := GVL_Cfg.GZ_UP;
        AxZ.Vel := GVL_Cfg.Z_VEL; AxZ.Acc := GVL_Cfg.Z_ACC;
        AxZ.MoveExec := TRUE;
        IF AxZ.Done THEN AxZ.MoveExec := FALSE; iSt := 21; END_IF
        IF AxZ.Error THEN iSt := 90; END_IF
    21: // step 2: IK + coordinated XY
        IK(xCart := tgtX, yCart := tgtY);
        IF NOT IK.Reachable THEN
            iSt := 0; Busy := FALSE; Error := TRUE;
            ErrorID := F_Err(GVL_Cfg.SS_GANTRY, GVL_Cfg.ERR_UNREACH);
        ELSE
            AxX.TargetPos := IK.xLin;     AxX.Vel := GVL_Cfg.G_VEL; AxX.Acc := GVL_Cfg.G_ACC;
            AxT.TargetPos := IK.thetaDeg; AxT.Vel := GVL_Cfg.T_VEL; AxT.Acc := GVL_Cfg.T_ACC;
            AxX.MoveExec := TRUE; AxT.MoveExec := TRUE;
            iSt := 22;
        END_IF
    22:
        IF AxX.Done AND AxT.Done THEN
            AxX.MoveExec := FALSE; AxT.MoveExec := FALSE; iSt := 23;
        END_IF
        IF AxX.Error OR AxT.Error THEN iSt := 90; END_IF
    23: // step 3: Z dip
        AxZ.TargetPos := zTarget; AxZ.MoveExec := TRUE;
        IF AxZ.Done THEN AxZ.MoveExec := FALSE; iSt := 24; END_IF
        IF AxZ.Error THEN iSt := 90; END_IF
    24: // step 4: arm grip/release; result checked next scan (Grip.Done may be stale this scan)
        IF cmdL.code = GVL_Cfg.MCMD_PICK THEN
            Grip.AcquireExec := TRUE;
        ELSE
            Grip.ReleaseExec := TRUE;
        END_IF
        iSt := 26;
    26: // wait gripper result
        IF Grip.Done THEN
            Grip.AcquireExec := FALSE; Grip.ReleaseExec := FALSE; iSt := 25;
        END_IF
        IF Grip.Error THEN
            Grip.AcquireExec := FALSE; Grip.ReleaseExec := FALSE;
            ErrorID := Grip.ErrorID; iSt := 90;
        END_IF
    25: // step 5: Z up -> done
        AxZ.TargetPos := GVL_Cfg.GZ_UP; AxZ.MoveExec := TRUE;
        IF AxZ.Done THEN
            AxZ.MoveExec := FALSE;
            iSt := 0; Busy := FALSE; Done := TRUE;
        END_IF
        IF AxZ.Error THEN iSt := 90; END_IF

    60: // PARK / SANITIZE: Z up then XY
        AxZ.TargetPos := GVL_Cfg.GZ_UP; AxZ.MoveExec := TRUE;
        IF AxZ.Done THEN AxZ.MoveExec := FALSE; iSt := 61; END_IF
        IF AxZ.Error THEN iSt := 90; END_IF
    61:
        IK(xCart := tgtX + GVL_Cfg.ARM_LEN, yCart := tgtY);  // park pose: arm at 0 deg
        AxX.TargetPos := tgtX;  AxX.Vel := GVL_Cfg.G_VEL; AxX.Acc := GVL_Cfg.G_ACC;
        AxT.TargetPos := 0.0;   AxT.Vel := GVL_Cfg.T_VEL; AxT.Acc := GVL_Cfg.T_ACC;
        AxX.MoveExec := TRUE; AxT.MoveExec := TRUE;
        iSt := 62;
    62:
        IF AxX.Done AND AxT.Done THEN
            AxX.MoveExec := FALSE; AxT.MoveExec := FALSE;
            iSt := 0; Busy := FALSE; Done := TRUE;
        END_IF
        IF AxX.Error OR AxT.Error THEN iSt := 90; END_IF

    90: // fault funnel
        AxX.MoveExec := FALSE; AxT.MoveExec := FALSE; AxZ.MoveExec := FALSE;
        Grip.AcquireExec := FALSE; Grip.ReleaseExec := FALSE;
        IF ErrorID = 0 THEN
            IF AxX.Error THEN ErrorID := AxX.ErrorID;
            ELSIF AxT.Error THEN ErrorID := AxT.ErrorID;
            ELSIF AxZ.Error THEN ErrorID := AxZ.ErrorID;
            ELSE ErrorID := F_Err(GVL_Cfg.SS_GANTRY, GVL_Cfg.ERR_DRIVE); END_IF
        END_IF
        iSt := 0; Busy := FALSE; Error := TRUE;
END_CASE
State := TO_UINT(iSt);

                  
END_FUNCTION_BLOCK

(* ============================================================ FB_GriddleCarousel — thin coordinator over FB_VfdIndex + pin FB_PneuActuator with the ROTATION PERMISSIVE interlock: all presses open + gantry parked + scraper parked (computed by PRG_JobExec, wired in PRG_Carousels). ActStation = index of the griddle currently AT THE LOAD STATION. Griddle g is at scrape station when ActStation = (g+2) MOD 4. Runs in T_App. ============================================================ *)
FUNCTION_BLOCK FB_GriddleCarousel
  VAR_INPUT
    Enable : BOOL;
    HomeExec : BOOL;
    GotoExec : BOOL;
    TargetStation : INT;
    RotatePermissive : BOOL;
    Abort : BOOL;
  END_VAR
  VAR_IN_OUT
    Vfd : FB_VfdIndex;
    Pin : FB_PneuActuator;
  END_VAR
  VAR_OUTPUT
    ActStation : INT;
    Homed : BOOL;
    Busy : BOOL;
    Done : BOOL;
    Error : BOOL;
    ErrorID : UDINT;
  END_VAR
  VAR
    rtGoto : R_TRIG;
    blocked : BOOL;
  END_VAR

                    rtGoto(CLK := GotoExec);

// wire pin actuator to indexing driver
Pin.Cmd          := Vfd.PinCmd;
Vfd.PinExtended  := Pin.Extended;
Vfd.PinRetracted := Pin.Retracted;

blocked := rtGoto.Q AND NOT RotatePermissive;
IF blocked THEN
    Error := TRUE;
    ErrorID := F_Err(GVL_Cfg.SS_GRID_CAR, GVL_Cfg.ERR_INTERLOCK);
END_IF

Vfd.Enable   := Enable;
Vfd.Abort    := Abort;
Vfd.HomeExec := HomeExec;
Vfd.GotoExec := GotoExec AND RotatePermissive;
Vfd.TargetStation := TargetStation;
Vfd.Bidirectional := TRUE;                 // shortest signed path

ActStation := Vfd.ActStation;
Homed := Vfd.Homed;
Busy  := Vfd.Busy;
Done  := Vfd.Done;
IF Vfd.Error THEN
    Error := TRUE; ErrorID := Vfd.ErrorID;
ELSIF NOT blocked THEN
    Error := FALSE; ErrorID := 0;
END_IF
IF Pin.Error THEN
    Error := TRUE; ErrorID := Pin.ErrorID;
END_IF

                  
END_FUNCTION_BLOCK

(* ============================================================ FB_Gripper — v1 stub over one pneumatic channel. INTERFACE IS FROZEN: swap internals when the real effector is designed. Owned pneu FB instance is external (GVL_Mech.fbPneuGrip), body called in PRG_Carousels; this FB only writes Cmd / reads status. Runs in T_Motion (with FB_Gantry). ============================================================ *)
FUNCTION_BLOCK FB_Gripper
  VAR_INPUT
    Sim : BOOL;
    AcquireExec : BOOL;  (* edge *)
    ReleaseExec : BOOL;
    iAcquired : BOOL;  (* patty-acquired feedback (sim: modeled) *)
    CycleMs : LREAL := 4.0;
  END_VAR
  VAR_IN_OUT
    Pneu : FB_PneuActuator;
  END_VAR
  VAR_OUTPUT
    Holding : BOOL;
    Busy : BOOL;
    Done : BOOL;
    Error : BOOL;
    ErrorID : UDINT;
  END_VAR
  VAR
    state : INT;
    rtA : R_TRIG;
    rtR : R_TRIG;
    tonTO : TON;
    acqEff : BOOL;
  END_VAR

                    rtA(CLK := AcquireExec);
rtR(CLK := ReleaseExec);
acqEff := (Sim AND Pneu.Extended) OR ((NOT Sim) AND iAcquired);

CASE state OF
    0:
        IF rtA.Q THEN Pneu.Cmd := TRUE;  state := 1; Busy := TRUE; Done := FALSE; tonTO(IN := FALSE); END_IF
        IF rtR.Q THEN Pneu.Cmd := FALSE; state := 2; Busy := TRUE; Done := FALSE; tonTO(IN := FALSE); END_IF
    1: // acquiring
        tonTO(IN := TRUE, PT := GVL_Cfg.TO_PNEU);
        IF Pneu.Extended AND acqEff THEN
            Holding := TRUE; state := 0; Busy := FALSE; Done := TRUE;
        ELSIF tonTO.Q THEN
            state := 0; Busy := FALSE; Error := TRUE;
            ErrorID := F_Err(GVL_Cfg.SS_GRIPPER, GVL_Cfg.ERR_TIMEOUT);
        END_IF
    2: // releasing
        tonTO(IN := TRUE, PT := GVL_Cfg.TO_PNEU);
        IF Pneu.Retracted THEN
            Holding := FALSE; state := 0; Busy := FALSE; Done := TRUE;
        ELSIF tonTO.Q THEN
            state := 0; Busy := FALSE; Error := TRUE;
            ErrorID := F_Err(GVL_Cfg.SS_GRIPPER, GVL_Cfg.ERR_TIMEOUT);
        END_IF
END_CASE


                  
END_FUNCTION_BLOCK

(* ============================================================ FB_HeatBank — supervises 8 FB_PidHeater zones: stagger tokens (inrush cap during ramp) + aggregate status. Call AFTER the heater bodies each T_App cycle (one-cycle token lag is fine). Zone map: griddle g -> zones 2g (top), 2g+1 (bottom). ============================================================ *)
FUNCTION_BLOCK FB_HeatBank
  VAR_INPUT
    Enable : BOOL;
  END_VAR
  VAR_IN_OUT
    Heaters : ARRAY[0..7] OF FB_PidHeater;
  END_VAR
  VAR_OUTPUT
    Token : ARRAY[0..7] OF BOOL;
    AllAtSet : BOOL;
    MaxDevC : LREAL;
    AnyTcErr : BOOL;
  END_VAR
  VAR
    z : INT;
    nRamping : INT;
    ramping : BOOL;
    dev : LREAL;
  END_VAR

                    nRamping := 0; AllAtSet := Enable; MaxDevC := 0.0; AnyTcErr := FALSE;
FOR z := 0 TO 7 DO
    ramping := (Heaters[z].Zone.setC - Heaters[z].Zone.actC) > 20.0;
    IF ramping THEN
        IF nRamping < GVL_Cfg.HEAT_MAX_STAGGER THEN
            Token[z] := TRUE; nRamping := nRamping + 1;
        ELSE
            Token[z] := FALSE;
        END_IF
    ELSE
        Token[z] := TRUE;   // regulation always allowed
    END_IF
    dev := ABS(Heaters[z].Zone.setC - Heaters[z].Zone.actC);
    IF dev > MaxDevC THEN MaxDevC := dev; END_IF
    IF NOT Heaters[z].Zone.atSet THEN AllAtSet := FALSE; END_IF
    IF Heaters[z].Error THEN AnyTcErr := TRUE; END_IF
END_FOR
IF NOT Enable THEN AllAtSet := FALSE; END_IF


                  
END_FUNCTION_BLOCK

(* ============================================================ FB_IKTransform — Cartesian (x,y) -> gantry (xLinear, thetaDeg). Model: carriage travels along X at y=0; arm of length ARM_LEN pivots on carriage: x = xLin + L*cos(theta), y = L*sin(theta) Solution: theta = ASIN(y/L) (elbow toward +x), xLin = x - L*cos. MILESTONE M1 GATE: validate over the full tray+griddle table in simulation (see TESTING_GUIDE TC-02) before any hardware motion. ============================================================ *)
FUNCTION_BLOCK FB_IKTransform
  VAR_INPUT
    xCart : LREAL;
    yCart : LREAL;
  END_VAR
  VAR_OUTPUT
    xLin : LREAL;
    thetaDeg : LREAL;
    Reachable : BOOL;
  END_VAR
  VAR
    rNorm : LREAL;
    thetaR : LREAL;
    PI_ : LREAL := 3.14159265358979;
  END_VAR

                    Reachable := FALSE;
IF ABS(yCart) > GVL_Cfg.ARM_LEN THEN RETURN; END_IF
rNorm := yCart / GVL_Cfg.ARM_LEN;
thetaR := ASIN(rNorm);
thetaDeg := thetaR * 180.0 / PI_;
xLin := xCart - GVL_Cfg.ARM_LEN * COS(thetaR);
Reachable := (xLin >= GVL_Cfg.GX_MIN) AND (xLin <= GVL_Cfg.GX_MAX)
         AND (thetaDeg >= GVL_Cfg.THETA_MIN) AND (thetaDeg <= GVL_Cfg.THETA_MAX);


                  
END_FUNCTION_BLOCK

(* ============================================================ FB_Press — one clamshell press. Wraps FB_PressDrive (paths: 0=OPEN 1=SMASH 2=HOLD). Executes the force/position profile: CLOSE->SMASH (smashDurS) -> BACK OFF to HOLD (light contact) -> stays HOLDING until MCMD_OPEN. Product-quality decision: never full force for the whole cook. Runs in T_App. Commands: MCMD_HOME(=open), MCMD_PROFILE, MCMD_OPEN. ============================================================ *)
FUNCTION_BLOCK FB_Press
  VAR_INPUT
    Enable : BOOL;
    Cmd : ST_MechCmd;
    CmdExec : BOOL;
    Abort : BOOL;
    Sim : BOOL;
    PressId : INT;
    Recipe : ST_Recipe;
    CycleMs : LREAL := 20.0;
  END_VAR
  VAR_IN_OUT
    Drv : FB_PressDrive;
  END_VAR
  VAR_OUTPUT
    Busy : BOOL;
    Done : BOOL;
    Error : BOOL;
    ErrorID : UDINT;
    State : UINT;
    IsOpen : BOOL;
    Holding : BOOL;
    DwellS : LREAL;  (* time at smash+hold, for HACCP *)
  END_VAR
  VAR
    iSt : INT;
    rtExec : R_TRIG;
    smashT : LREAL;
    scale : LREAL;
    tonTO : TON;  (* watchdog: any Busy state stuck -> labeled timeout *)
  END_VAR

                    rtExec(CLK := CmdExec);
scale := 1.0;
IF Sim THEN scale := GVL_Cfg.SIM_TIME_SCALE; END_IF

IF Abort THEN
    iSt := 0; Busy := FALSE;
    Drv.PathExec := FALSE; Drv.WriteParams := FALSE;
END_IF
IF Drv.Error AND (iSt <> 0) THEN
    iSt := 0; Busy := FALSE; Error := TRUE; ErrorID := Drv.ErrorID;
    Drv.PathExec := FALSE; Drv.WriteParams := FALSE;
END_IF

// watchdog — Busy states only (HOLDING has Busy=FALSE, so a long cook never trips it)
tonTO(IN := Busy, PT := GVL_Cfg.TO_MECH);
IF tonTO.Q AND Busy THEN
    iSt := 0; Busy := FALSE; Error := TRUE;
    ErrorID := F_Err(GVL_Cfg.SS_PRESS_0 + TO_UINT(PressId), GVL_Cfg.ERR_TIMEOUT);
    Drv.PathExec := FALSE; Drv.WriteParams := FALSE;
END_IF

CASE iSt OF
    0: // idle
        IF Enable AND rtExec.Q THEN
            Done := FALSE; Error := FALSE; ErrorID := 0;
            IF (Cmd.code = GVL_Cfg.MCMD_PROFILE) THEN
                IF NOT IsOpen THEN
                    Error := TRUE; ErrorID := F_Err(GVL_Cfg.SS_PRESS_0 + TO_UINT(PressId), GVL_Cfg.ERR_INTERLOCK);
                ELSE
                    DwellS := 0.0; smashT := 0.0;
                    // push PR positions (recipe + per-press calibration trim)
                    // to the drive before commanding motion
                    Drv.OpenPosMm  := GVL_Cfg.PRESS_OPEN_MM;
                    Drv.SmashPosMm := Recipe.smashPosMm + GVL_Par.pressTrimMm[PressId];
                    Drv.HoldPosMm  := Recipe.holdPosMm  + GVL_Par.pressTrimMm[PressId];
                    Drv.WriteParams := TRUE;
                    iSt := 5; Busy := TRUE; IsOpen := FALSE;
                END_IF
            ELSIF (Cmd.code = GVL_Cfg.MCMD_OPEN) OR (Cmd.code = GVL_Cfg.MCMD_HOME) THEN
                Drv.PathNo := 0; Drv.PathExec := TRUE;          // OPEN
                iSt := 30; Busy := TRUE; Holding := FALSE;
            ELSE
                Error := TRUE; ErrorID := F_Err(GVL_Cfg.SS_PRESS_0 + TO_UINT(PressId), GVL_Cfg.ERR_BAD_CMD);
            END_IF
        END_IF
    5: // wait for PR table confirmed in drive, then smash
        IF Drv.ParamsValid THEN
            Drv.WriteParams := FALSE;
            Drv.PathNo := 1; Drv.PathExec := TRUE;              // SMASH
            iSt := 10;
        ELSIF Drv.ParamErr THEN
            Drv.WriteParams := FALSE;
            iSt := 0; Busy := FALSE; Error := TRUE;
            ErrorID := F_Err(GVL_Cfg.SS_PRESS_0 + TO_UINT(PressId), GVL_Cfg.ERR_DRIVE);
        END_IF
    10: // closing to smash position
        IF Drv.Done THEN
            Drv.PathExec := FALSE; iSt := 11;
        END_IF
    11: // dwell at smash force/position
        smashT := smashT + CycleMs / 1000.0 * scale;
        DwellS := DwellS + CycleMs / 1000.0 * scale;
        IF smashT >= Recipe.smashDurS THEN
            Drv.PathNo := 2; Drv.PathExec := TRUE;              // BACK OFF -> HOLD
            iSt := 12;
        END_IF
    12:
        IF Drv.Done THEN
            Drv.PathExec := FALSE;
            iSt := 20; Busy := FALSE; Done := TRUE; Holding := TRUE;
        END_IF
    20: // HOLDING for cook duration (open on command)
        DwellS := DwellS + CycleMs / 1000.0 * scale;
        IF Enable AND rtExec.Q AND (Cmd.code = GVL_Cfg.MCMD_OPEN) THEN
            Done := FALSE;
            Drv.PathNo := 0; Drv.PathExec := TRUE;
            iSt := 30; Busy := TRUE; Holding := FALSE;
        END_IF
    30: // opening
        IF Drv.Done THEN
            Drv.PathExec := FALSE;
            iSt := 0; Busy := FALSE; Done := TRUE; IsOpen := TRUE;
        END_IF
END_CASE
State := TO_UINT(iSt);

                  
END_FUNCTION_BLOCK

(* ============================================================ FB_Refrigeration — compressor hysteresis + HACCP excursion timer. Runs in T_App. SIM: simple pulldown/heat-leak model. Excursion (> setpoint+0.5 C for FRIDGE_EXC_S) -> QUARANTINE flag (mapped by PRG_Alarms). ============================================================ *)
FUNCTION_BLOCK FB_Refrigeration
  VAR_INPUT
    Sim : BOOL;
    Enable : BOOL;
    iTempRaw : INT;  (* 0.1 degC *)
    CycleMs : LREAL := 20.0;
  END_VAR
  VAR_OUTPUT
    qCompressor : BOOL;
    ActC : LREAL;
    AtSet : BOOL;
    Excursion : BOOL;
    ErrorID : UDINT;
  END_VAR
  VAR
    simC : LREAL := 25.0;  (* pulldown from ambient at boot *)
    excT : LREAL;
    minRun : TON;
    minOff : TON;
    compReq : BOOL;
  END_VAR

                    IF Sim THEN
    IF qCompressor THEN
        simC := simC - 0.15 * (CycleMs / 1000.0) * GVL_Cfg.SIM_TIME_SCALE;
    ELSE
        simC := simC + 0.03 * (CycleMs / 1000.0) * GVL_Cfg.SIM_TIME_SCALE;
    END_IF
    simC := LIMIT(1.0, simC, 30.0);
    ActC := simC;
ELSE
    ActC := TO_LREAL(iTempRaw) / 10.0;
END_IF

// hysteresis with min run/stop (compressor protection)
IF ActC > GVL_Cfg.FRIDGE_SET_C + GVL_Cfg.FRIDGE_HYST_C THEN compReq := TRUE; END_IF
IF ActC < GVL_Cfg.FRIDGE_SET_C - GVL_Cfg.FRIDGE_HYST_C THEN compReq := FALSE; END_IF
minRun(IN := qCompressor, PT := T#60S);
minOff(IN := NOT qCompressor, PT := T#60S);
IF Enable THEN
    IF compReq AND (minOff.Q OR Sim) THEN qCompressor := TRUE; END_IF
    IF (NOT compReq) AND (minRun.Q OR Sim) THEN qCompressor := FALSE; END_IF
ELSE
    qCompressor := FALSE;
END_IF

AtSet := ActC <= GVL_Cfg.FRIDGE_SET_C + 1.0;

IF Enable AND (ActC > GVL_Cfg.FRIDGE_SET_C + 0.5) AND AtSet = FALSE AND (GVL_Sts.mode = E_MachMode.RUN) THEN
    excT := excT + CycleMs / 1000.0 * GVL_Cfg.SIM_TIME_SCALE;
ELSE
    excT := 0.0;
END_IF
Excursion := excT >= GVL_Cfg.FRIDGE_EXC_S;
IF Excursion THEN
    ErrorID := F_Err(GVL_Cfg.SS_REFRIG, GVL_Cfg.ERR_SENSOR);
END_IF

                  
END_FUNCTION_BLOCK

(* ============================================================ FB_Scraper — sweep mechanism. Commands: MCMD_HOME, MCMD_PARK, MCMD_SWEEP(p1=strokeIdx 0..2). One SWEEP = position at row, Z engage, X sweep across, Z up, return. Caller (JobExec) guarantees the interlock: griddle at scrape station, clamshell open, press retracted. Runs in T_Motion. ============================================================ *)
FUNCTION_BLOCK FB_Scraper
  VAR_INPUT
    Enable : BOOL;
    Cmd : ST_MechCmd;
    CmdExec : BOOL;
    Abort : BOOL;
    Sim : BOOL;
    InterlockOk : BOOL;  (* from JobExec: safe to engage *)
  END_VAR
  VAR_IN_OUT
    AxX : FB_AxisCtrl;
    AxY : FB_AxisCtrl;
    AxZ : FB_AxisCtrl;
  END_VAR
  VAR_OUTPUT
    Busy : BOOL;
    Done : BOOL;
    Error : BOOL;
    ErrorID : UDINT;
    State : UINT;
    Homed : BOOL;
    Parked : BOOL;
  END_VAR
  VAR
    iSt : INT;
    rtExec : R_TRIG;
    stroke : INT;
    tonTO : TON;
  END_VAR

                    rtExec(CLK := CmdExec);
IF Abort THEN
    iSt := 0; Busy := FALSE;
    AxX.MoveExec := FALSE; AxY.MoveExec := FALSE; AxZ.MoveExec := FALSE;
    AxX.HomeExec := FALSE; AxY.HomeExec := FALSE; AxZ.HomeExec := FALSE;
END_IF
Homed  := AxX.Sts.homed AND AxY.Sts.homed AND AxZ.Sts.homed;
Parked := Homed AND (iSt = 0);

tonTO(IN := Busy, PT := GVL_Cfg.TO_MECH);
IF tonTO.Q AND Busy THEN
    iSt := 0; Busy := FALSE; Error := TRUE;
    ErrorID := F_Err(GVL_Cfg.SS_SCRAPER, GVL_Cfg.ERR_TIMEOUT);
END_IF

CASE iSt OF
    0:
        IF Enable AND rtExec.Q THEN
            Done := FALSE; Error := FALSE; ErrorID := 0;
            CASE Cmd.code OF
                1:  (* MCMD_HOME *)  iSt := 10; Busy := TRUE;
                30: (* MCMD_SWEEP *)
                    stroke := TO_INT(Cmd.p1);
                    IF (stroke < 0) OR (stroke >= GVL_Cfg.SC_STROKES) THEN
                        Error := TRUE; ErrorID := F_Err(GVL_Cfg.SS_SCRAPER, GVL_Cfg.ERR_BAD_CMD);
                    ELSIF NOT InterlockOk THEN
                        Error := TRUE; ErrorID := F_Err(GVL_Cfg.SS_SCRAPER, GVL_Cfg.ERR_INTERLOCK);
                    ELSE
                        iSt := 20; Busy := TRUE;
                    END_IF
                2:  (* MCMD_PARK *)  iSt := 60; Busy := TRUE;
            ELSE
                Error := TRUE; ErrorID := F_Err(GVL_Cfg.SS_SCRAPER, GVL_Cfg.ERR_BAD_CMD);
            END_CASE
        END_IF
    10: // HOME: Z first
        AxZ.HomeExec := TRUE;
        IF AxZ.Sts.homed THEN AxZ.HomeExec := FALSE; iSt := 11; END_IF
    11:
        AxX.HomeExec := TRUE;
        IF AxX.Sts.homed THEN AxX.HomeExec := FALSE; iSt := 12; END_IF
    12:
        AxY.HomeExec := TRUE;
        IF AxY.Sts.homed THEN
            AxY.HomeExec := FALSE; iSt := 0; Busy := FALSE; Done := TRUE;
        END_IF
    20: // position at stroke start, Z up
        AxZ.TargetPos := GVL_Cfg.SC_UP_Z; AxZ.Vel := GVL_Cfg.Z_VEL; AxZ.Acc := GVL_Cfg.Z_ACC;
        AxZ.MoveExec := TRUE;
        IF AxZ.Done THEN AxZ.MoveExec := FALSE; iSt := 21; END_IF
        IF AxZ.Error THEN iSt := 90; END_IF
    21:
        AxX.TargetPos := GVL_Cfg.SC_SWEEP_X0; AxX.Vel := GVL_Cfg.S_VEL; AxX.Acc := GVL_Cfg.S_ACC;
        AxY.TargetPos := GVL_Cfg.SC_ROW_Y[stroke]; AxY.Vel := GVL_Cfg.S_VEL; AxY.Acc := GVL_Cfg.S_ACC;
        AxX.MoveExec := TRUE; AxY.MoveExec := TRUE;
        iSt := 22;
    22:
        IF AxX.Done AND AxY.Done THEN
            AxX.MoveExec := FALSE; AxY.MoveExec := FALSE; iSt := 23;
        END_IF
        IF AxX.Error OR AxY.Error THEN iSt := 90; END_IF
    23: // engage blade
        AxZ.TargetPos := GVL_Cfg.SC_ENGAGE_Z; AxZ.MoveExec := TRUE;
        IF AxZ.Done THEN AxZ.MoveExec := FALSE; iSt := 24; END_IF
        IF AxZ.Error THEN iSt := 90; END_IF
    24: // sweep across
        AxX.TargetPos := GVL_Cfg.SC_SWEEP_X1; AxX.MoveExec := TRUE;
        IF AxX.Done THEN AxX.MoveExec := FALSE; iSt := 25; END_IF
        IF AxX.Error THEN iSt := 90; END_IF
    25: // blade up -> done
        AxZ.TargetPos := GVL_Cfg.SC_UP_Z; AxZ.MoveExec := TRUE;
        IF AxZ.Done THEN
            AxZ.MoveExec := FALSE; iSt := 0; Busy := FALSE; Done := TRUE;
        END_IF
        IF AxZ.Error THEN iSt := 90; END_IF
    60: // PARK
        AxZ.TargetPos := GVL_Cfg.SC_UP_Z; AxZ.MoveExec := TRUE;
        IF AxZ.Done THEN AxZ.MoveExec := FALSE; iSt := 61; END_IF
        IF AxZ.Error THEN iSt := 90; END_IF
    61:
        AxX.TargetPos := 0.0; AxY.TargetPos := 0.0;
        AxX.MoveExec := TRUE; AxY.MoveExec := TRUE;
        IF AxX.Done AND AxY.Done THEN
            AxX.MoveExec := FALSE; AxY.MoveExec := FALSE;
            iSt := 0; Busy := FALSE; Done := TRUE;
        END_IF
        IF AxX.Error OR AxY.Error THEN iSt := 90; END_IF
    90:
        AxX.MoveExec := FALSE; AxY.MoveExec := FALSE; AxZ.MoveExec := FALSE;
        IF ErrorID = 0 THEN
            IF AxX.Error THEN ErrorID := AxX.ErrorID;
            ELSIF AxY.Error THEN ErrorID := AxY.ErrorID;
            ELSIF AxZ.Error THEN ErrorID := AxZ.ErrorID;
            ELSE ErrorID := F_Err(GVL_Cfg.SS_SCRAPER, GVL_Cfg.ERR_DRIVE); END_IF
        END_IF
        iSt := 0; Busy := FALSE; Error := TRUE;
END_CASE
State := TO_UINT(iSt);

                  
END_FUNCTION_BLOCK

(* ============================================================ FB_GriddleTracker — per-griddle state + cook timers + HACCP record emission. Runs in T_App (called from PRG_JobExec's PRG). ScrapeDue fires at cookTime - SCRAPE_GUARD_S so the coordinator can stage the scraper. NewHaccp is a LATCHED flag: set here, cleared by the consumer (PRG_HACCP, slower task) after reading. ============================================================ *)
FUNCTION_BLOCK FB_GriddleTracker
  VAR_INPUT
    Sim : BOOL;
    CycleMs : LREAL := 20.0;
    SetLoading : BOOL;  (* griddle being loaded *)
    GIdxA : INT;  (* griddle being loaded *)
    StartCook : BOOL;
    GIdxB : INT;
    ItemB : UINT;
    CountB : INT;
    BatchB : UDINT;
    ScrapeStart : BOOL;
    GIdxC : INT;
    ScrapeDone : BOOL;
    GIdxD : INT;
    SetFault : BOOL;
    GIdxE : INT;
    HaccpAck : BOOL;  (* consumer (PRG_HACCP) sets after reading the record *)
  END_VAR
  VAR_OUTPUT
    aG : ARRAY[0..3] OF ST_GriddleSts;
    ScrapeDue : BOOL;
    ScrapeDueG : INT := -1;
    NewHaccp : BOOL;
    HaccpRec : ST_HaccpRec;
  END_VAR
  VAR
    rtL : R_TRIG;
    rtS : R_TRIG;
    rtP : R_TRIG;
    rtD : R_TRIG;
    rtF : R_TRIG;
    g : INT;
    dtS : LREAL;
    rec : ST_HaccpRec;
    startS : ARRAY[0..3] OF UDINT;
  END_VAR

                    dtS := CycleMs / 1000.0;
IF Sim THEN dtS := dtS * GVL_Cfg.SIM_TIME_SCALE; END_IF
rtL(CLK := SetLoading);  rtS(CLK := StartCook);  rtP(CLK := ScrapeStart);
rtD(CLK := ScrapeDone);  rtF(CLK := SetFault);
// NewHaccp stays latched until the consumer acks it (T_Comms is 5x
// slower than T_App; a 1-cycle pulse would get lost)
IF HaccpAck THEN NewHaccp := FALSE; END_IF

IF rtL.Q AND (GIdxA >= 0) AND (GIdxA <= 3) THEN
    aG[GIdxA].state := TO_UINT(E_GriddleState.LOADING);
END_IF
IF rtS.Q AND (GIdxB >= 0) AND (GIdxB <= 3) THEN
    aG[GIdxB].state := TO_UINT(E_GriddleState.COOKING);
    aG[GIdxB].item  := ItemB;
    aG[GIdxB].count := CountB;
    aG[GIdxB].batchId := BatchB;
    aG[GIdxB].cookElapsedS := 0.0;
    startS[GIdxB] := GVL_Sts.uptimeS;
END_IF
IF rtP.Q AND (GIdxC >= 0) AND (GIdxC <= 3) THEN
    aG[GIdxC].state := TO_UINT(E_GriddleState.SCRAPING);
END_IF
IF rtD.Q AND (GIdxD >= 0) AND (GIdxD <= 3) THEN
    // emit HACCP record, then empty the griddle
    rec.batchId    := aG[GIdxD].batchId;
    rec.item       := aG[GIdxD].item;
    rec.griddleId  := GIdxD;
    rec.platenTopC := GVL_Sts.aHeat[2 * GIdxD].actC;
    rec.platenBotC := GVL_Sts.aHeat[2 * GIdxD + 1].actC;
    rec.cookS      := aG[GIdxD].cookElapsedS;
    rec.tStartS    := startS[GIdxD];
    rec.tEndS      := GVL_Sts.uptimeS;
    IF (rec.platenTopC < GVL_Par.aRecipe[rec.item].platenSetC - 15.0)
       OR (rec.cookS < GVL_Par.aRecipe[rec.item].cookTimeS - 2.0) THEN
        rec.result := 1;    // QUARANTINE
    ELSE
        rec.result := 0;
    END_IF
    HaccpRec := rec; NewHaccp := TRUE;
    aG[GIdxD].state := TO_UINT(E_GriddleState.EMPTY);
    aG[GIdxD].item := 0; aG[GIdxD].count := 0; aG[GIdxD].cookElapsedS := 0.0;
END_IF
IF rtF.Q AND (GIdxE >= 0) AND (GIdxE <= 3) THEN
    aG[GIdxE].state := TO_UINT(E_GriddleState.FAULTED);
END_IF

// cook timers + due flag
ScrapeDue := FALSE; ScrapeDueG := -1;
FOR g := 0 TO 3 DO
    IF aG[g].state = TO_UINT(E_GriddleState.COOKING) THEN
        aG[g].cookElapsedS := aG[g].cookElapsedS + dtS;
        IF aG[g].cookElapsedS >= GVL_Par.aRecipe[aG[g].item].cookTimeS - GVL_Cfg.SCRAPE_GUARD_S THEN
            aG[g].state := TO_UINT(E_GriddleState.READY_TO_SCRAPE);
        END_IF
    END_IF
    IF (aG[g].state = TO_UINT(E_GriddleState.READY_TO_SCRAPE)) AND (ScrapeDueG < 0) THEN
        ScrapeDue := TRUE; ScrapeDueG := g;
    END_IF
    // keep elapsed counting until scraped (for HACCP truth)
    IF aG[g].state = TO_UINT(E_GriddleState.READY_TO_SCRAPE)
       OR aG[g].state = TO_UINT(E_GriddleState.SCRAPING) THEN
        aG[g].cookElapsedS := aG[g].cookElapsedS + dtS;
    END_IF
END_FOR

                  
END_FUNCTION_BLOCK

(* ============================================================ FB_HomingManager — collision-safe machine homing (spec 8.3): presses OPEN -> gantry -> scraper -> fork -> griddle carousel -> fridge carousel. Runs in T_App (called by PRG_Supervisor, which executes BEFORE PRG_Carousels in the task list). ============================================================ *)
FUNCTION_BLOCK FB_HomingManager
  VAR_INPUT
    Exec : BOOL;
    Abort : BOOL;
  END_VAR
  VAR_IN_OUT
    Presses : ARRAY[0..3] OF FB_Press;
    Gantry : FB_Gantry;
    Scraper : FB_Scraper;
    Fork : FB_Fork;
    GridCar : FB_GriddleCarousel;
    FridgeCar : FB_FridgeCarousel;
  END_VAR
  VAR_OUTPUT
    Busy : BOOL;
    Done : BOOL;
    Error : BOOL;
    ErrorID : UDINT;
    Step : UINT;
  END_VAR
  VAR
    iSt : INT;
    i : INT;
    rtExec : R_TRIG;
    tonTO : TON;
    allOpen : BOOL;
  END_VAR

                    rtExec(CLK := Exec);
IF Abort THEN iSt := 0; Busy := FALSE; END_IF
tonTO(IN := Busy, PT := T#120S);
IF tonTO.Q AND Busy THEN
    iSt := 0; Busy := FALSE; Error := TRUE;
    ErrorID := F_Err(GVL_Cfg.SS_HOMING, GVL_Cfg.ERR_TIMEOUT);
END_IF

CASE iSt OF
    0:
        IF rtExec.Q THEN
            Done := FALSE; Error := FALSE; ErrorID := 0;
            iSt := 10; Busy := TRUE;
        END_IF
    10: // command all presses OPEN
        FOR i := 0 TO 3 DO
            Presses[i].Cmd.code := GVL_Cfg.MCMD_OPEN;
            Presses[i].CmdExec := TRUE;
        END_FOR
        iSt := 11;
    11:
        allOpen := TRUE;
        FOR i := 0 TO 3 DO
            IF NOT Presses[i].IsOpen THEN allOpen := FALSE; END_IF
            IF Presses[i].Error THEN iSt := 90; ErrorID := Presses[i].ErrorID; END_IF
        END_FOR
        IF allOpen AND (iSt = 11) THEN
            FOR i := 0 TO 3 DO Presses[i].CmdExec := FALSE; END_FOR
            iSt := 20;
        END_IF
    20: // gantry
        Gantry.Cmd.code := GVL_Cfg.MCMD_HOME; Gantry.CmdExec := TRUE;
        iSt := 21;
    21:
        IF Gantry.Done AND Gantry.Homed THEN Gantry.CmdExec := FALSE; iSt := 30; END_IF
        IF Gantry.Error THEN ErrorID := Gantry.ErrorID; iSt := 90; END_IF
    30: // scraper
        Scraper.Cmd.code := GVL_Cfg.MCMD_HOME; Scraper.CmdExec := TRUE;
        iSt := 31;
    31:
        IF Scraper.Done AND Scraper.Homed THEN Scraper.CmdExec := FALSE; iSt := 40; END_IF
        IF Scraper.Error THEN ErrorID := Scraper.ErrorID; iSt := 90; END_IF
    40: // fork
        Fork.Cmd.code := GVL_Cfg.MCMD_HOME; Fork.CmdExec := TRUE;
        iSt := 41;
    41:
        IF Fork.Done AND Fork.Homed THEN Fork.CmdExec := FALSE; iSt := 50; END_IF
        IF Fork.Error THEN ErrorID := Fork.ErrorID; iSt := 90; END_IF
    50: // griddle carousel
        GridCar.HomeExec := TRUE;
        iSt := 51;
    51:
        IF GridCar.Homed THEN GridCar.HomeExec := FALSE; iSt := 60; END_IF
        IF GridCar.Error THEN ErrorID := GridCar.ErrorID; iSt := 90; END_IF
    60: // fridge carousel
        FridgeCar.HomeExec := TRUE;
        iSt := 61;
    61:
        IF FridgeCar.Homed THEN
            FridgeCar.HomeExec := FALSE;
            iSt := 0; Busy := FALSE; Done := TRUE;
        END_IF
        IF FridgeCar.Error THEN ErrorID := FridgeCar.ErrorID; iSt := 90; END_IF
    90:
        Gantry.CmdExec := FALSE; Scraper.CmdExec := FALSE; Fork.CmdExec := FALSE;
        GridCar.HomeExec := FALSE; FridgeCar.HomeExec := FALSE;
        FOR i := 0 TO 3 DO Presses[i].CmdExec := FALSE; END_FOR
        iSt := 0; Busy := FALSE; Error := TRUE;
END_CASE
Step := TO_UINT(iSt);


                  
END_FUNCTION_BLOCK

(* ============================================================ FB_JobQueue — ring buffer of ST_PattyJob (size 64). ============================================================ *)
FUNCTION_BLOCK FB_JobQueue
  VAR_INPUT
    PushExec : BOOL;
    JobIn : ST_PattyJob;
    PopExec : BOOL;
    ClearExec : BOOL;
  END_VAR
  VAR_OUTPUT
    JobOut : ST_PattyJob;
    Count : INT;
    Full : BOOL;
    Empty : BOOL;
    PopOk : BOOL;
  END_VAR
  VAR
    buf : ARRAY[0..63] OF ST_PattyJob;
    head : INT;  (* next write *)
    tail : INT;  (* next read *)
    rtPush : R_TRIG;
    rtPop : R_TRIG;
    rtClr : R_TRIG;
  END_VAR

                    rtPush(CLK := PushExec);
rtPop(CLK := PopExec);
rtClr(CLK := ClearExec);
IF rtClr.Q THEN head := 0; tail := 0; Count := 0; END_IF
Full  := Count >= 64;
Empty := Count = 0;
PopOk := FALSE;
IF rtPush.Q AND NOT Full THEN
    buf[head] := JobIn;
    head := (head + 1) MOD 64;
    Count := Count + 1;
END_IF
IF rtPop.Q AND NOT Empty THEN
    JobOut := buf[tail];
    tail := (tail + 1) MOD 64;
    Count := Count - 1;
    PopOk := TRUE;
END_IF


                  
END_FUNCTION_BLOCK

(* ============================================================ PRG_JobExec — executes Gateway primitives (T_App, after Supervisor). Enforces ORDER SAFETY only; scheduling policy is the Gateway's. Autonomous behavior: if a cook completes and the Gateway is silent (or no command pending), scrape locally — patties never burn waiting for a dead PC. In testMode this program idles (PRG_Test has authority). Primitive sub-sequences use numbered CASE states: 100+ FETCH_TRAY 200+ LOAD_GRIDDLE 300+ SCRAPE 400+ RETURN_TRAY ============================================================ *)
PROGRAM PRG_JobExec
  VAR
    iSt : INT;
    g : INT;  (* target griddle *)
    item : UINT;
    count : INT;
    level : INT;
    face : INT;
    i : INT;  (* patty loop index *)
    trayIdx : INT;
    batchSeq : UDINT;
    autoScrape : BOOL;
    rotPerm : BOOL;
    tonGw : TON;
    tonStep : TON;
    scrapeStroke : INT;
  END_VAR

                    
// ---- Gateway liveness ----
tonGw(IN := TRUE, PT := T#10S);   // re-armed by comms on heartbeat change
IF GVL_Cmd.gwAlive THEN tonGw(IN := FALSE); tonGw(IN := TRUE); END_IF
GVL_Sts.gwSilent := NOT GVL_Cmd.gwAlive;

// ---- rotation permissive for the griddle carousel ----
rotPerm := TRUE;
FOR i := 0 TO 3 DO
    // presses may rotate while HOLDING (they travel with the disc) but
    // never mid-motion
    IF GVL_Mech.fbPress[i].Busy THEN rotPerm := FALSE; END_IF
END_FOR
IF NOT GVL_Mech.fbGantry.Parked  THEN rotPerm := FALSE; END_IF
IF NOT GVL_Mech.fbScraper.Parked THEN rotPerm := FALSE; END_IF
GVL_Mech.fbGridCar.RotatePermissive := rotPerm;

// ---- tracker body (always runs) ----
GVL_Mech.fbTracker(Sim := GVL_Cfg.SIM_MODE);
GVL_Sts.aGriddle := GVL_Mech.fbTracker.aG;

// clear tracker command pulses after body call
GVL_Mech.fbTracker.SetLoading  := FALSE;
GVL_Mech.fbTracker.StartCook   := FALSE;
GVL_Mech.fbTracker.ScrapeStart := FALSE;
GVL_Mech.fbTracker.ScrapeDone  := FALSE;

IF GVL_Cmd.testMode THEN RETURN; END_IF
IF GVL_Sts.mode <> E_MachMode.RUN THEN
    IF iSt <> 0 THEN iSt := 0; END_IF   // mode fell out mid-primitive: mechanisms abort via Supervisor
    RETURN;
END_IF

tonStep(IN := iSt <> 0, PT := T#300S);
IF tonStep.Q AND (iSt <> 0) THEN
    GVL_Cmd.gwAck.error := TRUE;
    GVL_Cmd.gwAck.errorId := F_Err(GVL_Cfg.SS_JOBEXEC, GVL_Cfg.ERR_TIMEOUT);
    GVL_Cmd.gwAck.busy := FALSE; GVL_Cmd.gwPending := FALSE;
    iSt := 0;
END_IF

CASE iSt OF
    0: // ---- dispatch ----
        autoScrape := FALSE;
        IF GVL_Cmd.gwPending THEN
            IF GVL_Cmd.gwCmd.code = GVL_Cfg.CMD_FETCH_TRAY THEN
                item := TO_UINT(GVL_Cmd.gwCmd.p1); level := TO_INT(GVL_Cmd.gwCmd.p2); face := TO_INT(GVL_Cmd.gwCmd.p3);
                iSt := 100;
            ELSIF GVL_Cmd.gwCmd.code = GVL_Cfg.CMD_LOAD_GRIDDLE THEN
                g := TO_INT(GVL_Cmd.gwCmd.p1); count := TO_INT(GVL_Cmd.gwCmd.p2); item := TO_UINT(GVL_Cmd.gwCmd.p3);
                IF (g < 0) OR (g > 3) OR (count < 1) OR (count > GVL_Cfg.PATTIES_PER_GRIDDLE)
                   OR (GVL_Sts.aGriddle[g].state <> TO_UINT(E_GriddleState.EMPTY))
                   OR (NOT GVL_Sts.tray.inChamber) OR (GVL_Sts.tray.remaining < count) THEN
                    GVL_Cmd.gwAck.error := TRUE;
                    GVL_Cmd.gwAck.errorId := F_Err(GVL_Cfg.SS_JOBEXEC, GVL_Cfg.ERR_BAD_CMD);
                    GVL_Cmd.gwAck.busy := FALSE; GVL_Cmd.gwPending := FALSE;
                ELSE
                    iSt := 200;
                END_IF
            ELSIF GVL_Cmd.gwCmd.code = GVL_Cfg.CMD_SCRAPE THEN
                g := TO_INT(GVL_Cmd.gwCmd.p1);
                iSt := 300;
            ELSIF GVL_Cmd.gwCmd.code = GVL_Cfg.CMD_RETURN_TRAY THEN
                level := TO_INT(GVL_Cmd.gwCmd.p1); face := TO_INT(GVL_Cmd.gwCmd.p2);
                iSt := 400;
            ELSIF GVL_Cmd.gwCmd.code = GVL_Cfg.CMD_CLEAN_MODE THEN
                GVL_Cmd.reqClean := TRUE;
                GVL_Cmd.gwAck.done := TRUE; GVL_Cmd.gwAck.busy := FALSE; GVL_Cmd.gwPending := FALSE;
            ELSIF GVL_Cmd.gwCmd.code = GVL_Cfg.CMD_ABORT THEN
                GVL_Cmd.reqStop := TRUE;
                GVL_Cmd.gwAck.done := TRUE; GVL_Cmd.gwAck.busy := FALSE; GVL_Cmd.gwPending := FALSE;
            ELSE
                GVL_Cmd.gwAck.error := TRUE;
                GVL_Cmd.gwAck.errorId := F_Err(GVL_Cfg.SS_JOBEXEC, GVL_Cfg.ERR_BAD_CMD);
                GVL_Cmd.gwAck.busy := FALSE; GVL_Cmd.gwPending := FALSE;
            END_IF
        ELSIF GVL_Mech.fbTracker.ScrapeDue AND GVL_Sts.gwSilent THEN
            // AUTONOMOUS FINISH: gateway dead, cook done -> scrape locally
            g := GVL_Mech.fbTracker.ScrapeDueG;
            autoScrape := TRUE;
            iSt := 300;
        END_IF

    // ================= FETCH_TRAY =================
    100: // rotate fridge column to face (fork must be retracted/parked)
        GVL_Mech.fbFridgeCar.Permissive := NOT GVL_Mech.fbFork.Busy;
        GVL_Mech.fbFridgeCar.TargetFace := face;
        GVL_Mech.fbFridgeCar.GotoExec := TRUE;
        iSt := 101;
    101:
        IF GVL_Mech.fbFridgeCar.Done OR (GVL_Mech.fbFridgeCar.ActFace = face) THEN
            GVL_Mech.fbFridgeCar.GotoExec := FALSE; iSt := 102;
        ELSIF GVL_Mech.fbFridgeCar.Error THEN iSt := 900;
        END_IF
    102: // open fridge-side gate
        GVL_Mech.fbAirlock.ReqFridgeOpen := TRUE;
        IF GVL_Mech.fbAirlock.FridgeOpen THEN iSt := 103; END_IF
        IF GVL_Mech.fbAirlock.Error THEN iSt := 900; END_IF
    103: // fork fetch
        GVL_Mech.fbFork.Cmd.code := GVL_Cfg.MCMD_FETCH;
        GVL_Mech.fbFork.Cmd.p1 := TO_LREAL(level);
        GVL_Mech.fbFork.CmdExec := TRUE;
        iSt := 104;
    104:
        IF GVL_Mech.fbFork.Done AND GVL_Mech.fbFork.TrayHeld THEN
            GVL_Mech.fbFork.CmdExec := FALSE; iSt := 105;
        ELSIF GVL_Mech.fbFork.Error THEN
            GVL_Mech.fbFork.CmdExec := FALSE; iSt := 900;
        END_IF
    105: // close gate; publish tray info
        GVL_Mech.fbAirlock.ReqFridgeOpen := FALSE;
        IF GVL_Mech.fbAirlock.ChamberSealed THEN
            GVL_Sts.tray.item := item;
            GVL_Sts.tray.remaining := GVL_Cfg.PATTIES_PER_TRAY;
            GVL_Sts.tray.level := level; GVL_Sts.tray.face := face;
            GVL_Sts.tray.inChamber := TRUE;
            iSt := 990;
        END_IF

    // ================= LOAD_GRIDDLE =================
    200: // bring griddle g to load station
        GVL_Mech.fbTracker.SetLoading := TRUE; GVL_Mech.fbTracker.GIdxA := g;
        GVL_Mech.fbGridCar.TargetStation := g;
        GVL_Mech.fbGridCar.GotoExec := TRUE;
        iSt := 201;
    201:
        IF GVL_Mech.fbGridCar.Done OR (GVL_Mech.fbGridCar.ActStation = g) THEN
            GVL_Mech.fbGridCar.GotoExec := FALSE; iSt := 202;
        ELSIF GVL_Mech.fbGridCar.Error THEN iSt := 900;
        END_IF
    202: // open chamber gate (fridge side must be sealed)
        GVL_Mech.fbAirlock.ReqChamberOpen := TRUE;
        IF GVL_Mech.fbAirlock.ChamberOpen THEN i := 0; iSt := 210; END_IF
        IF GVL_Mech.fbAirlock.Error THEN iSt := 900; END_IF
    210: // pick patty i from tray
        trayIdx := GVL_Cfg.PATTIES_PER_TRAY - GVL_Sts.tray.remaining;
        GVL_Mech.fbGantry.Cmd.code := GVL_Cfg.MCMD_PICK;
        GVL_Mech.fbGantry.Cmd.p1 := TO_LREAL(trayIdx);
        GVL_Mech.fbGantry.CmdExec := TRUE;
        iSt := 211;
    211:
        IF GVL_Mech.fbGantry.Done THEN
            GVL_Mech.fbGantry.CmdExec := FALSE; iSt := 212;
        ELSIF GVL_Mech.fbGantry.Error THEN
            GVL_Mech.fbGantry.CmdExec := FALSE; iSt := 900;
        END_IF
    212: // place on griddle slot i
        GVL_Mech.fbGantry.Cmd.code := GVL_Cfg.MCMD_PLACE;
        GVL_Mech.fbGantry.Cmd.p1 := TO_LREAL(i);
        GVL_Mech.fbGantry.CmdExec := TRUE;
        iSt := 213;
    213:
        IF GVL_Mech.fbGantry.Done THEN
            GVL_Mech.fbGantry.CmdExec := FALSE;
            GVL_Sts.pattyOnGriddle[g, i] := TRUE;
            GVL_Sts.tray.remaining := GVL_Sts.tray.remaining - 1;
            i := i + 1;
            IF i >= count THEN iSt := 220; ELSE iSt := 210; END_IF
        ELSIF GVL_Mech.fbGantry.Error THEN
            GVL_Mech.fbGantry.CmdExec := FALSE; iSt := 900;
        END_IF
    220: // park gantry, close chamber
        GVL_Mech.fbGantry.Cmd.code := GVL_Cfg.MCMD_PARK;
        GVL_Mech.fbGantry.CmdExec := TRUE;
        iSt := 221;
    221:
        IF GVL_Mech.fbGantry.Done THEN
            GVL_Mech.fbGantry.CmdExec := FALSE;
            GVL_Mech.fbAirlock.ReqChamberOpen := FALSE;
            iSt := 222;
        ELSIF GVL_Mech.fbGantry.Error THEN
            GVL_Mech.fbGantry.CmdExec := FALSE; iSt := 900;
        END_IF
    222:
        IF GVL_Mech.fbAirlock.ChamberSealed THEN iSt := 230; END_IF
    230: // run press profile + start cook clock
        GVL_Mech.fbPress[g].Recipe := GVL_Par.aRecipe[item];
        GVL_Mech.fbPress[g].Cmd.code := GVL_Cfg.MCMD_PROFILE;
        GVL_Mech.fbPress[g].CmdExec := TRUE;
        iSt := 231;
    231:
        IF GVL_Mech.fbPress[g].Holding THEN
            GVL_Mech.fbPress[g].CmdExec := FALSE;
            batchSeq := batchSeq + 1;
            GVL_Mech.fbTracker.StartCook := TRUE;
            GVL_Mech.fbTracker.GIdxB := g;
            GVL_Mech.fbTracker.ItemB := item;
            GVL_Mech.fbTracker.CountB := count;
            GVL_Mech.fbTracker.BatchB := batchSeq;
            iSt := 990;
        ELSIF GVL_Mech.fbPress[g].Error THEN
            GVL_Mech.fbPress[g].CmdExec := FALSE; iSt := 900;
        END_IF

    // ================= SCRAPE =================
    300: // open press g first
        GVL_Mech.fbTracker.ScrapeStart := TRUE; GVL_Mech.fbTracker.GIdxC := g;
        GVL_Mech.fbPress[g].Cmd.code := GVL_Cfg.MCMD_OPEN;
        GVL_Mech.fbPress[g].CmdExec := TRUE;
        iSt := 301;
    301:
        IF GVL_Mech.fbPress[g].IsOpen THEN
            GVL_Mech.fbPress[g].CmdExec := FALSE; iSt := 302;
        ELSIF GVL_Mech.fbPress[g].Error THEN
            GVL_Mech.fbPress[g].CmdExec := FALSE; iSt := 900;
        END_IF
    302: // rotate griddle g to scrape station
        GVL_Mech.fbGridCar.TargetStation := (g + 2) MOD 4;
        GVL_Mech.fbGridCar.GotoExec := TRUE;
        iSt := 303;
    303:
        IF (GVL_Mech.fbGridCar.Done OR (GVL_Mech.fbGridCar.ActStation = (g + 2) MOD 4))
           AND NOT GVL_Mech.fbGridCar.Busy THEN   // arrival can be reported while still settling
            GVL_Mech.fbGridCar.GotoExec := FALSE;
            scrapeStroke := 0; iSt := 310;
        ELSIF GVL_Mech.fbGridCar.Error THEN iSt := 900;
        END_IF
    310: // sweep strokes — only command when the interlock is actually satisfied
        GVL_Mech.fbScraper.InterlockOk := GVL_Mech.fbPress[g].IsOpen AND NOT GVL_Mech.fbGridCar.Busy;
        IF GVL_Mech.fbScraper.InterlockOk THEN
            GVL_Mech.fbScraper.Cmd.code := GVL_Cfg.MCMD_SWEEP;
            GVL_Mech.fbScraper.Cmd.p1 := TO_LREAL(scrapeStroke);
            GVL_Mech.fbScraper.CmdExec := TRUE;
            iSt := 311;
        END_IF
    311:
        IF GVL_Mech.fbScraper.Done THEN
            GVL_Mech.fbScraper.CmdExec := FALSE;
            scrapeStroke := scrapeStroke + 1;
            IF scrapeStroke >= GVL_Cfg.SC_STROKES THEN iSt := 320; ELSE iSt := 310; END_IF
        ELSIF GVL_Mech.fbScraper.Error THEN
            GVL_Mech.fbScraper.CmdExec := FALSE; iSt := 900;
        END_IF
    320: // park scraper, finish batch bookkeeping
        GVL_Mech.fbScraper.Cmd.code := GVL_Cfg.MCMD_PARK;
        GVL_Mech.fbScraper.CmdExec := TRUE;
        iSt := 321;
    321:
        IF GVL_Mech.fbScraper.Done THEN
            GVL_Mech.fbScraper.CmdExec := FALSE;
            FOR i := 0 TO 5 DO GVL_Sts.pattyOnGriddle[g, i] := FALSE; END_FOR
            GVL_Mech.fbTracker.ScrapeDone := TRUE; GVL_Mech.fbTracker.GIdxD := g;
            iSt := 990;
        ELSIF GVL_Mech.fbScraper.Error THEN
            GVL_Mech.fbScraper.CmdExec := FALSE; iSt := 900;
        END_IF

    // ================= RETURN_TRAY =================
    400:
        GVL_Mech.fbAirlock.ReqFridgeOpen := TRUE;
        IF GVL_Mech.fbAirlock.FridgeOpen THEN iSt := 401; END_IF
        IF GVL_Mech.fbAirlock.Error THEN iSt := 900; END_IF
    401:
        GVL_Mech.fbFork.Cmd.code := GVL_Cfg.MCMD_RETURN;
        GVL_Mech.fbFork.Cmd.p1 := TO_LREAL(level);
        GVL_Mech.fbFork.CmdExec := TRUE;
        iSt := 402;
    402:
        IF GVL_Mech.fbFork.Done THEN
            GVL_Mech.fbFork.CmdExec := FALSE;
            GVL_Mech.fbAirlock.ReqFridgeOpen := FALSE;
            GVL_Sts.tray.inChamber := FALSE;
            iSt := 403;
        ELSIF GVL_Mech.fbFork.Error THEN
            GVL_Mech.fbFork.CmdExec := FALSE; iSt := 900;
        END_IF
    403:
        IF GVL_Mech.fbAirlock.ChamberSealed THEN iSt := 990; END_IF

    // ================= exits =================
    900: // primitive failed
        IF NOT autoScrape THEN
            GVL_Cmd.gwAck.error := TRUE;
            GVL_Cmd.gwAck.errorId := F_Err(GVL_Cfg.SS_JOBEXEC, GVL_Cfg.ERR_DRIVE);
            GVL_Cmd.gwAck.busy := FALSE; GVL_Cmd.gwPending := FALSE;
        END_IF
        iSt := 0;
    990: // primitive done
        IF NOT autoScrape THEN
            GVL_Cmd.gwAck.done := TRUE;
            GVL_Cmd.gwAck.busy := FALSE; GVL_Cmd.gwPending := FALSE;
        END_IF
        iSt := 0;
END_CASE


                  
END_PROGRAM

(* ============================================================ PRG_Supervisor — machine mode state machine (T_App, runs FIRST among coordinators). Owns: mode transitions, enable distribution, abort broadcast, homing orchestration, clean-mode thermal gate. Safety is only MONITORED here (GVL_Sts.safetyOk). ============================================================ *)
PROGRAM PRG_Supervisor
  VAR
    rtStart : R_TRIG;
    rtStop : R_TRIG;
    rtReset : R_TRIG;
    rtClean : R_TRIG;
    z : INT;
    coolOk : BOOL;
    firstScan : BOOL := TRUE;
  END_VAR

                    // effective safety status
GVL_Sts.safetyOk := GVL_Cfg.SIM_MODE OR GVL_IO.iSafetyOk;

rtStart(CLK := GVL_Cmd.reqStart);
rtStop (CLK := GVL_Cmd.reqStop);
rtReset(CLK := GVL_Cmd.reqReset);
rtClean(CLK := GVL_Cmd.reqClean);

// defaults each scan
GVL_Sts.resetPulse := FALSE;

// global overrides
IF NOT GVL_Sts.safetyOk THEN
    GVL_Sts.mode := E_MachMode.ESTOP;
END_IF
IF GVL_Alm.reqMachStop AND (GVL_Sts.mode <> E_MachMode.ESTOP) THEN
    GVL_Sts.mode := E_MachMode.FAULT;
END_IF

CASE GVL_Sts.mode OF
    E_MachMode.BOOT:
        GVL_Sts.enMotion := FALSE; GVL_Sts.enProcess := FALSE;
        GVL_Sts.abortAll := FALSE;
        IF GVL_Sts.safetyOk AND NOT firstScan THEN
            GVL_Sts.resetPulse := TRUE;
            GVL_Mech.fbHoming.Exec := TRUE;
            GVL_Sts.mode := E_MachMode.HOMING;
        END_IF

    E_MachMode.HOMING:
        GVL_Sts.enMotion := TRUE; GVL_Sts.enProcess := FALSE;
        IF GVL_Mech.fbHoming.Done THEN
            GVL_Mech.fbHoming.Exec := FALSE;
            GVL_Sts.mode := E_MachMode.READY;
        ELSIF GVL_Mech.fbHoming.Error THEN
            GVL_Mech.fbHoming.Exec := FALSE;
            GVL_Sts.mode := E_MachMode.FAULT;
        END_IF

    E_MachMode.READY:
        GVL_Sts.enMotion := TRUE; GVL_Sts.enProcess := TRUE;   // heat-up + pulldown
        IF GVL_Alm.reqZoneStop THEN
            GVL_Sts.mode := E_MachMode.FAULT;
        ELSIF rtStart.Q AND GVL_Sts.heatAtSet AND GVL_Sts.fridgeAtSet AND GVL_Sts.allHomed THEN
            GVL_Sts.mode := E_MachMode.RUN;
        END_IF

    E_MachMode.RUN:
        GVL_Sts.enMotion := TRUE; GVL_Sts.enProcess := TRUE;
        IF GVL_Alm.reqZoneStop THEN
            GVL_Sts.mode := E_MachMode.FAULT;
        ELSIF rtStop.Q THEN
            GVL_Sts.mode := E_MachMode.READY;      // finish-in-place is JobExec's job
        ELSIF rtClean.Q AND (GVL_Mech.fbQueue.Empty) THEN
            GVL_Sts.mode := E_MachMode.CLEAN;
        END_IF

    E_MachMode.CLEAN:
        GVL_Sts.enMotion := FALSE;                  // motion locked for operator
        GVL_Sts.enProcess := FALSE;                 // heaters off -> cool down
        coolOk := TRUE;
        FOR z := 0 TO 7 DO
            IF GVL_Sts.aHeat[z].actC >= 60.0 THEN coolOk := FALSE; END_IF
        END_FOR
        GVL_Sts.cleanCoolOk := coolOk;
        IF rtStart.Q AND coolOk THEN                // operator confirms clean done
            GVL_Sts.resetPulse := TRUE;
            GVL_Mech.fbHoming.Exec := TRUE;
            GVL_Sts.mode := E_MachMode.HOMING;
        END_IF

    E_MachMode.FAULT:
        GVL_Sts.enMotion := FALSE; GVL_Sts.enProcess := FALSE;
        GVL_Sts.abortAll := TRUE;
        IF rtReset.Q AND (NOT GVL_Alm.reqMachStop) AND (NOT GVL_Alm.reqZoneStop) THEN
            GVL_Sts.abortAll := FALSE;
            GVL_Sts.resetPulse := TRUE;
            GVL_Mech.fbHoming.Exec := TRUE;
            GVL_Sts.mode := E_MachMode.HOMING;
        END_IF

    E_MachMode.ESTOP:
        GVL_Sts.enMotion := FALSE; GVL_Sts.enProcess := FALSE;
        GVL_Sts.abortAll := TRUE;
        IF GVL_Sts.safetyOk AND rtReset.Q THEN
            GVL_Sts.abortAll := FALSE;
            GVL_Sts.resetPulse := TRUE;
            GVL_Mech.fbHoming.Exec := TRUE;
            GVL_Sts.mode := E_MachMode.HOMING;
        END_IF
END_CASE
firstScan := FALSE;

// homing manager body (same task, before PRG_Carousels)
GVL_Mech.fbHoming(
    Abort     := GVL_Sts.abortAll,
    Presses   := GVL_Mech.fbPress,
    Gantry    := GVL_Mech.fbGantry,
    Scraper   := GVL_Mech.fbScraper,
    Fork      := GVL_Mech.fbFork,
    GridCar   := GVL_Mech.fbGridCar,
    FridgeCar := GVL_Mech.fbFridgeCar);

// aggregates
GVL_Sts.allHomed := GVL_Mech.fbGantry.Homed AND GVL_Mech.fbScraper.Homed
                AND GVL_Mech.fbFork.Homed AND GVL_Mech.fbGridCar.Homed
                AND GVL_Mech.fbFridgeCar.Homed;
GVL_Sts.heatAtSet   := GVL_Mech.fbHeatBank.AllAtSet;
GVL_Sts.fridgeAtSet := GVL_Mech.fbRefrig.AtSet;
GVL_Sts.fridgeActC  := GVL_Mech.fbRefrig.ActC;


                  
END_PROGRAM

(* ============================================================ PRG_Alarms — central alarm manager (T_App, runs LAST). Raises on the RISING edge of each source Error (so an acked alarm doesn't re-raise from a still-latched source; sources clear their Error on the next command latch / axis reset). Class map (spec sec.13): MACHINE_STOP : fork brake/drive integrity ZONE_STOP : axis/drive faults, pin mismatch, TC fault, airlock violation, mechanism timeouts QUARANTINE : fridge excursion, short-cook (via PRG_HACCP) INFO : gateway silent ============================================================ *)
PROGRAM PRG_Alarms
  VAR
    i : INT;
    n : INT;
    worst : UINT;
    rtAck : R_TRIG;
    rtGw : R_TRIG;
    rtGan : R_TRIG;
    rtScr : R_TRIG;
    rtFrk : R_TRIG;
    rtGC : R_TRIG;
    rtFC : R_TRIG;
    rtAir : R_TRIG;
    rtExc : R_TRIG;
    rtPress : ARRAY[0..3] OF R_TRIG;
    rtHeat : ARRAY[0..7] OF R_TRIG;
  END_VAR

                    // ---- collect (edge-raised) ----
rtFrk(CLK := GVL_Mech.fbFork.Error);
IF rtFrk.Q THEN
    IF SHR(GVL_Mech.fbFork.ErrorID, 16) = TO_UDINT(GVL_Cfg.SS_FORK_Z) THEN
        F_RaiseAlarm(GVL_Mech.fbFork.ErrorID, TO_UINT(E_FaultClass.MACHINE_STOP));
    ELSE
        F_RaiseAlarm(GVL_Mech.fbFork.ErrorID, TO_UINT(E_FaultClass.ZONE_STOP));
    END_IF
END_IF
rtGan(CLK := GVL_Mech.fbGantry.Error);
IF rtGan.Q THEN F_RaiseAlarm(GVL_Mech.fbGantry.ErrorID, TO_UINT(E_FaultClass.ZONE_STOP)); END_IF
rtScr(CLK := GVL_Mech.fbScraper.Error);
IF rtScr.Q THEN F_RaiseAlarm(GVL_Mech.fbScraper.ErrorID, TO_UINT(E_FaultClass.ZONE_STOP)); END_IF
rtGC(CLK := GVL_Mech.fbGridCar.Error);
IF rtGC.Q THEN F_RaiseAlarm(GVL_Mech.fbGridCar.ErrorID, TO_UINT(E_FaultClass.ZONE_STOP)); END_IF
rtFC(CLK := GVL_Mech.fbFridgeCar.Error);
IF rtFC.Q THEN F_RaiseAlarm(GVL_Mech.fbFridgeCar.ErrorID, TO_UINT(E_FaultClass.ZONE_STOP)); END_IF
rtAir(CLK := GVL_Mech.fbAirlock.Error);
IF rtAir.Q THEN F_RaiseAlarm(GVL_Mech.fbAirlock.ErrorID, TO_UINT(E_FaultClass.ZONE_STOP)); END_IF
FOR i := 0 TO 3 DO
    rtPress[i](CLK := GVL_Mech.fbPress[i].Error);
    IF rtPress[i].Q THEN
        F_RaiseAlarm(GVL_Mech.fbPress[i].ErrorID, TO_UINT(E_FaultClass.ZONE_STOP));
    END_IF
END_FOR
FOR i := 0 TO 7 DO
    rtHeat[i](CLK := GVL_Mech.fbHeater[i].Error);
    IF rtHeat[i].Q THEN
        F_RaiseAlarm(GVL_Mech.fbHeater[i].ErrorID, TO_UINT(E_FaultClass.ZONE_STOP));
    END_IF
END_FOR
rtExc(CLK := GVL_Mech.fbRefrig.Excursion);
IF rtExc.Q THEN
    F_RaiseAlarm(GVL_Mech.fbRefrig.ErrorID, TO_UINT(E_FaultClass.QUARANTINE));
END_IF
rtGw(CLK := GVL_Sts.gwSilent AND (GVL_Sts.mode = E_MachMode.RUN) AND NOT GVL_Cmd.testMode);
IF rtGw.Q THEN
    F_RaiseAlarm(F_Err(GVL_Cfg.SS_GWCOMMS, GVL_Cfg.ERR_TIMEOUT), TO_UINT(E_FaultClass.INFO));
END_IF

// ---- ack / clear ----
rtAck(CLK := GVL_Cmd.reqAckAll);
n := 0; worst := 0;
FOR i := 0 TO 63 DO
    IF GVL_Alm.aActive[i].active THEN
        IF rtAck.Q THEN GVL_Alm.aActive[i].acked := TRUE; END_IF
        IF GVL_Alm.aActive[i].acked THEN
            GVL_Alm.aActive[i].active := FALSE;
        ELSE
            n := n + 1;
            IF GVL_Alm.aActive[i].class > worst THEN worst := GVL_Alm.aActive[i].class; END_IF
        END_IF
    END_IF
END_FOR
GVL_Alm.nActive := n;
GVL_Alm.worstClass := worst;
GVL_Alm.reqZoneStop := worst >= TO_UINT(E_FaultClass.ZONE_STOP);
GVL_Alm.reqMachStop := worst >= TO_UINT(E_FaultClass.MACHINE_STOP);
GVL_Sts.activeAlarms := n;


                  
END_PROGRAM

(* ============================================================ PRG_GatewayComms — Modbus-TCP register map + seq/ack handshake (T_Comms, 100 ms). PLC is Modbus TCP slave; Gateway reads/writes the %MW images declared in GVL_Cmd. Register map (holding registers, 1 reg = 1 WORD): CMD %MW0..9 : [0]=seq [1]=code [2..3]=p1 lo/hi [4..5]=p2 [6..7]=p3 [8]=p4(lo only) [9]=gwHeartbeat ACK %MW10..15 : [10]=seqEcho [11]=flags(b0 busy b1 done b2 err) [12..13]=errorId lo/hi [14]=plc heartbeat STS %MW20..99 : see packing below PAR %MW500.. : [500]=item [501]=cookTimeS*10 [502]=setC*10 [503]=applyToggle (change -> apply, READY only) ============================================================ *)
PROGRAM PRG_GatewayComms
  VAR
    lastSeq : UINT;
    lastHb : UINT;
    hbAge : INT;
    flags : WORD;
    z : INT;
    gIdx : INT;
    parToggle : WORD;
    lastParTog : WORD;
    itemP : INT;
    cookP : LREAL;
    setP : LREAL;
  END_VAR

                    // ---------- decode command ----------
GVL_Cmd.gwCmd.seq  := GVL_Cmd.mbCmdRegs[0];
GVL_Cmd.gwCmd.code := GVL_Cmd.mbCmdRegs[1];
GVL_Cmd.gwCmd.p1 := WORD_TO_DINT(GVL_Cmd.mbCmdRegs[2]) + SHL(WORD_TO_DINT(GVL_Cmd.mbCmdRegs[3]), 16);
GVL_Cmd.gwCmd.p2 := WORD_TO_DINT(GVL_Cmd.mbCmdRegs[4]) + SHL(WORD_TO_DINT(GVL_Cmd.mbCmdRegs[5]), 16);
GVL_Cmd.gwCmd.p3 := WORD_TO_DINT(GVL_Cmd.mbCmdRegs[6]) + SHL(WORD_TO_DINT(GVL_Cmd.mbCmdRegs[7]), 16);
GVL_Cmd.gwCmd.p4 := WORD_TO_DINT(GVL_Cmd.mbCmdRegs[8]);
GVL_Cmd.gwHeartbeatIn := GVL_Cmd.mbCmdRegs[9];

// ---------- gateway liveness (heartbeat must CHANGE) ----------
IF GVL_Cmd.gwHeartbeatIn <> lastHb THEN
    lastHb := GVL_Cmd.gwHeartbeatIn; hbAge := 0;
ELSE
    hbAge := MIN(hbAge + 1, 32000);
END_IF
GVL_Cmd.gwAlive := hbAge < 100;   // 100 * 100 ms = 10 s

// ---------- new command latch ----------
IF (GVL_Cmd.gwCmd.seq <> lastSeq) AND (GVL_Cmd.gwCmd.seq <> 0) THEN
    IF GVL_Cmd.gwPending OR GVL_Cmd.gwAck.busy THEN
        // reject: still executing previous
        GVL_Cmd.gwAck.error := TRUE;
        GVL_Cmd.gwAck.errorId := F_Err(GVL_Cfg.SS_GWCOMMS, GVL_Cfg.ERR_BUSY);
        lastSeq := GVL_Cmd.gwCmd.seq;
        GVL_Cmd.gwAck.seqEcho := lastSeq;
    ELSIF GVL_Cmd.testMode THEN
        GVL_Cmd.gwAck.error := TRUE;
        GVL_Cmd.gwAck.errorId := F_Err(GVL_Cfg.SS_GWCOMMS, GVL_Cfg.ERR_INTERLOCK);
        lastSeq := GVL_Cmd.gwCmd.seq;
        GVL_Cmd.gwAck.seqEcho := lastSeq;
    ELSE
        lastSeq := GVL_Cmd.gwCmd.seq;
        GVL_Cmd.gwAck.seqEcho := lastSeq;
        GVL_Cmd.gwAck.busy := TRUE;
        GVL_Cmd.gwAck.done := FALSE;
        GVL_Cmd.gwAck.error := FALSE;
        GVL_Cmd.gwAck.errorId := 0;
        GVL_Cmd.gwPending := TRUE;
    END_IF
END_IF

// ---------- pack ack ----------
flags := 0;
IF GVL_Cmd.gwAck.busy  THEN flags := flags OR 16#0001; END_IF
IF GVL_Cmd.gwAck.done  THEN flags := flags OR 16#0002; END_IF
IF GVL_Cmd.gwAck.error THEN flags := flags OR 16#0004; END_IF
GVL_Cmd.mbAckRegs[0] := GVL_Cmd.gwAck.seqEcho;
GVL_Cmd.mbAckRegs[1] := flags;
GVL_Cmd.mbAckRegs[2] := DWORD_TO_WORD(GVL_Cmd.gwAck.errorId AND 16#FFFF);
GVL_Cmd.mbAckRegs[3] := DWORD_TO_WORD(SHR(GVL_Cmd.gwAck.errorId, 16));
GVL_Sts.heartbeat := GVL_Sts.heartbeat + 1;
GVL_Cmd.mbAckRegs[4] := GVL_Sts.heartbeat;

// ---------- pack status ----------
GVL_Cmd.mbStsRegs[0] := TO_WORD(TO_UINT(GVL_Sts.mode));
GVL_Cmd.mbStsRegs[1] := BOOL_TO_WORD(GVL_Sts.allHomed)
                      + SHL(BOOL_TO_WORD(GVL_Sts.heatAtSet), 1)
                      + SHL(BOOL_TO_WORD(GVL_Sts.fridgeAtSet), 2)
                      + SHL(BOOL_TO_WORD(GVL_Sts.gwSilent), 3)
                      + SHL(BOOL_TO_WORD(GVL_Cmd.testMode), 4);
FOR z := 0 TO 7 DO
    GVL_Cmd.mbStsRegs[10 + z] := TO_WORD(LREAL_TO_INT(GVL_Sts.aHeat[z].actC * 10.0));
END_FOR
GVL_Cmd.mbStsRegs[18] := TO_WORD(LREAL_TO_INT(GVL_Sts.fridgeActC * 10.0));
FOR gIdx := 0 TO 3 DO
    GVL_Cmd.mbStsRegs[20 + 3 * gIdx]     := TO_WORD(GVL_Sts.aGriddle[gIdx].state);
    GVL_Cmd.mbStsRegs[20 + 3 * gIdx + 1] := TO_WORD(GVL_Sts.aGriddle[gIdx].item);
    GVL_Cmd.mbStsRegs[20 + 3 * gIdx + 2] := TO_WORD(LREAL_TO_INT(GVL_Sts.aGriddle[gIdx].cookElapsedS));
END_FOR
GVL_Cmd.mbStsRegs[32] := TO_WORD(TO_UINT(GVL_Sts.tray.remaining));
GVL_Cmd.mbStsRegs[33] := BOOL_TO_WORD(GVL_Sts.tray.inChamber);
GVL_Cmd.mbStsRegs[34] := TO_WORD(TO_UINT(GVL_Sts.activeAlarms));
GVL_Cmd.mbStsRegs[35] := TO_WORD(TO_UINT(GVL_Sts.carGridStation + 1));
GVL_Cmd.mbStsRegs[36] := UDINT_TO_WORD(GVL_Sts.haccpCount AND 16#FFFF);
// latest HACCP record snapshot (Gateway drains richer log later — TODO ring window)
GVL_Cmd.mbStsRegs[60] := UDINT_TO_WORD(GVL_Sts.lastHaccp.batchId AND 16#FFFF);
GVL_Cmd.mbStsRegs[61] := TO_WORD(GVL_Sts.lastHaccp.item);
GVL_Cmd.mbStsRegs[62] := TO_WORD(TO_UINT(GVL_Sts.lastHaccp.griddleId));
GVL_Cmd.mbStsRegs[63] := TO_WORD(LREAL_TO_INT(GVL_Sts.lastHaccp.platenTopC * 10.0));
GVL_Cmd.mbStsRegs[64] := TO_WORD(LREAL_TO_INT(GVL_Sts.lastHaccp.platenBotC * 10.0));
GVL_Cmd.mbStsRegs[65] := TO_WORD(LREAL_TO_INT(GVL_Sts.lastHaccp.cookS));
GVL_Cmd.mbStsRegs[66] := TO_WORD(GVL_Sts.lastHaccp.result);

// ---------- recipe writes (READY only, bounds-checked) ----------
parToggle := GVL_Cmd.mbParRegs[3];
IF (parToggle <> lastParTog) AND (GVL_Sts.mode = E_MachMode.READY) THEN
    lastParTog := parToggle;
    itemP := WORD_TO_INT(GVL_Cmd.mbParRegs[0]);
    cookP := TO_LREAL(WORD_TO_INT(GVL_Cmd.mbParRegs[1])) / 10.0;
    setP  := TO_LREAL(WORD_TO_INT(GVL_Cmd.mbParRegs[2])) / 10.0;
    IF (itemP >= 1) AND (itemP <= 4)
       AND (cookP >= 20.0) AND (cookP <= 300.0)
       AND (setP >= 120.0) AND (setP <= 230.0) THEN
        GVL_Par.aRecipe[itemP].cookTimeS  := cookP;
        GVL_Par.aRecipe[itemP].platenSetC := setP;
    END_IF
END_IF


                  
END_PROGRAM

(* ============================================================ PRG_HACCP — cook record collector (T_Comms). RETAIN ring of 512 records (> one shift). Gateway currently reads the LATEST record snapshot from STS regs; full drain protocol via read pointer is a marked TODO for Gateway integration (M4). ============================================================ *)
PROGRAM PRG_HACCP
  VAR RETAIN
    ring : ARRAY[0..511] OF ST_HaccpRec;
    head : INT;
  END_VAR

                    IF GVL_Mech.fbTracker.NewHaccp AND NOT GVL_Mech.fbTracker.HaccpAck THEN
    ring[head] := GVL_Mech.fbTracker.HaccpRec;
    head := (head + 1) MOD 512;
    GVL_Sts.haccpCount := GVL_Sts.haccpCount + 1;
    GVL_Sts.lastHaccp := GVL_Mech.fbTracker.HaccpRec;
    IF GVL_Mech.fbTracker.HaccpRec.result = 1 THEN
        F_RaiseAlarm(F_Err(GVL_Cfg.SS_JOBEXEC, GVL_Cfg.ERR_SENSOR),
                     TO_UINT(E_FaultClass.QUARANTINE));
    END_IF
    GVL_Mech.fbTracker.HaccpAck := TRUE;       // tracker clears NewHaccp
ELSIF NOT GVL_Mech.fbTracker.NewHaccp THEN
    GVL_Mech.fbTracker.HaccpAck := FALSE;      // handshake complete, re-arm
END_IF

                  
END_PROGRAM

(* ============================================================ PRG_HMI — HMI request edges + password-gated jog (T_Comms). Buttons arrive as GVL_Cmd.hmi* (mapped to HMI tags at site). NOTE: in the SFC/LD refactor this POU's edge networks become LD rungs one-per-button (technician-facing). ============================================================ *)
PROGRAM PRG_HMI
  VAR
    rtStart : R_TRIG;
    rtStop : R_TRIG;
    rtReset : R_TRIG;
    rtAck : R_TRIG;
    rtClean : R_TRIG;
    jogPermit : BOOL;
    jogStep : LREAL;
    tonJog : TON;
    MAINT_PIN : UINT := 2468;  (* TODO site-specific, move to secure store *)
    rtRecW : R_TRIG;
    rtTrimW : R_TRIG;
    recOk : BOOL;
    recIt : INT;
    recV : LREAL;
    trimP : INT;
    bJogP : BOOL;  (* jog levels (direct var OR HMI register bit) *)
    bJogM : BOOL;  (* jog levels (direct var OR HMI register bit) *)
    wFlags : WORD;
    it2 : INT;
    z2 : INT;
    base : INT;
  END_VAR

